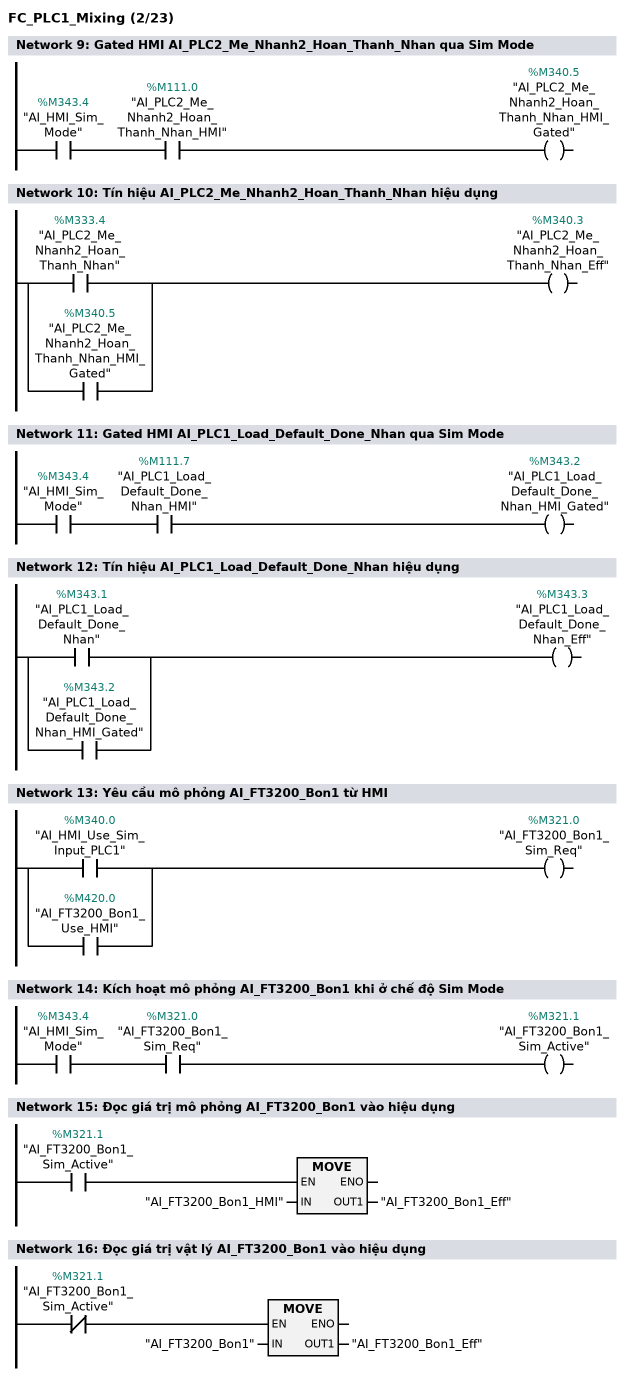
   RUNG wire#powerrail
      Contact( "AI_HMI_Sim_Mode" )
      Contact( "AI_PLC2_Me_Nhanh2_Hoan_Thanh_Nhan_HMI" )
      Coil( "AI_PLC2_Me_Nhanh2_Hoan_Thanh_Nhan_HMI_Gated" )
   END_RUNG
   // the same network as SCL:
   "AI_PLC2_Me_Nhanh2_Hoan_Thanh_Nhan_HMI_Gated" := "AI_HMI_Sim_Mode" AND "AI_PLC2_Me_Nhanh2_Hoan_Thanh_Nhan_HMI";
END_REGION

REGION Network 10: Tín hiệu AI_PLC2_Me_Nhanh2_Hoan_Thanh_Nhan hiệu dụng
   RUNG wire#powerrail
      Contact( "AI_PLC2_Me_Nhanh2_Hoan_Thanh_Nhan" )
      wire#w1
      Coil( "AI_PLC2_Me_Nhanh2_Hoan_Thanh_Nhan_Eff" )
   END_RUNG
   RUNG wire#powerrail
      Contact( "AI_PLC2_Me_Nhanh2_Hoan_Thanh_Nhan_HMI_Gated" )
   END_RUNG wire#w1
   // the same network as SCL:
   "AI_PLC2_Me_Nhanh2_Hoan_Thanh_Nhan_Eff" := "AI_PLC2_Me_Nhanh2_Hoan_Thanh_Nhan" OR "AI_PLC2_Me_Nhanh2_Hoan_Thanh_Nhan_HMI_Gated";
END_REGION

REGION Network 11: Gated HMI AI_PLC1_Load_Default_Done_Nhan qua Sim Mode
   RUNG wire#powerrail
      Contact( "AI_HMI_Sim_Mode" )
      Contact( "AI_PLC1_Load_Default_Done_Nhan_HMI" )
      Coil( "AI_PLC1_Load_Default_Done_Nhan_HMI_Gated" )
   END_RUNG
   // the same network as SCL:
   "AI_PLC1_Load_Default_Done_Nhan_HMI_Gated" := "AI_HMI_Sim_Mode" AND "AI_PLC1_Load_Default_Done_Nhan_HMI";
END_REGION

REGION Network 12: Tín hiệu AI_PLC1_Load_Default_Done_Nhan hiệu dụng
   RUNG wire#powerrail
      Contact( "AI_PLC1_Load_Default_Done_Nhan" )
      wire#w1
      Coil( "AI_PLC1_Load_Default_Done_Nhan_Eff" )
   END_RUNG
   RUNG wire#powerrail
      Contact( "AI_PLC1_Load_Default_Done_Nhan_HMI_Gated" )
   END_RUNG wire#w1
   // the same network as SCL:
   "AI_PLC1_Load_Default_Done_Nhan_Eff" := "AI_PLC1_Load_Default_Done_Nhan" OR "AI_PLC1_Load_Default_Done_Nhan_HMI_Gated";
END_REGION

REGION Network 13: Yêu cầu mô phỏng AI_FT3200_Bon1 từ HMI
   RUNG wire#powerrail
      Contact( "AI_HMI_Use_Sim_Input_PLC1" )
      wire#w1
      Coil( "AI_FT3200_Bon1_Sim_Req" )
   END_RUNG
   RUNG wire#powerrail
      Contact( "AI_FT3200_Bon1_Use_HMI" )
   END_RUNG wire#w1
   // the same network as SCL:
   "AI_FT3200_Bon1_Sim_Req" := "AI_HMI_Use_Sim_Input_PLC1" OR "AI_FT3200_Bon1_Use_HMI";
END_REGION

REGION Network 14: Kích hoạt mô phỏng AI_FT3200_Bon1 khi ở chế độ Sim Mode
   RUNG wire#powerrail
      Contact( "AI_HMI_Sim_Mode" )
      Contact( "AI_FT3200_Bon1_Sim_Req" )
      Coil( "AI_FT3200_Bon1_Sim_Active" )
   END_RUNG
   // the same network as SCL:
   "AI_FT3200_Bon1_Sim_Active" := "AI_HMI_Sim_Mode" AND "AI_FT3200_Bon1_Sim_Req";
END_REGION

REGION Network 15: Đọc giá trị mô phỏng AI_FT3200_Bon1 vào hiệu dụng
   RUNG wire#powerrail
      Contact( "AI_FT3200_Bon1_Sim_Active" )
      { S7_GenerateENO := "TRUE" } Move(in := "AI_FT3200_Bon1_HMI", out1 => "AI_FT3200_Bon1_Eff")
   END_RUNG
   // the same network as SCL:
   IF "AI_FT3200_Bon1_Sim_Active" THEN "AI_FT3200_Bon1_Eff" := "AI_FT3200_Bon1_HMI"; END_IF;
END_REGION

REGION Network 16: Đọc giá trị vật lý AI_FT3200_Bon1 vào hiệu dụng
   RUNG wire#powerrail
      I_Contact( "AI_FT3200_Bon1_Sim_Active" )
      { S7_GenerateENO := "TRUE" } Move(in := "AI_FT3200_Bon1", out1 => "AI_FT3200_Bon1_Eff")
   END_RUNG
   // the same network as SCL:
   IF NOT "AI_FT3200_Bon1_Sim_Active" THEN "AI_FT3200_Bon1_Eff" := "AI_FT3200_Bon1"; END_IF;
END_REGION

REGION Network 17: Yêu cầu mô phỏng AI_FQ3200_Bon1 từ HMI
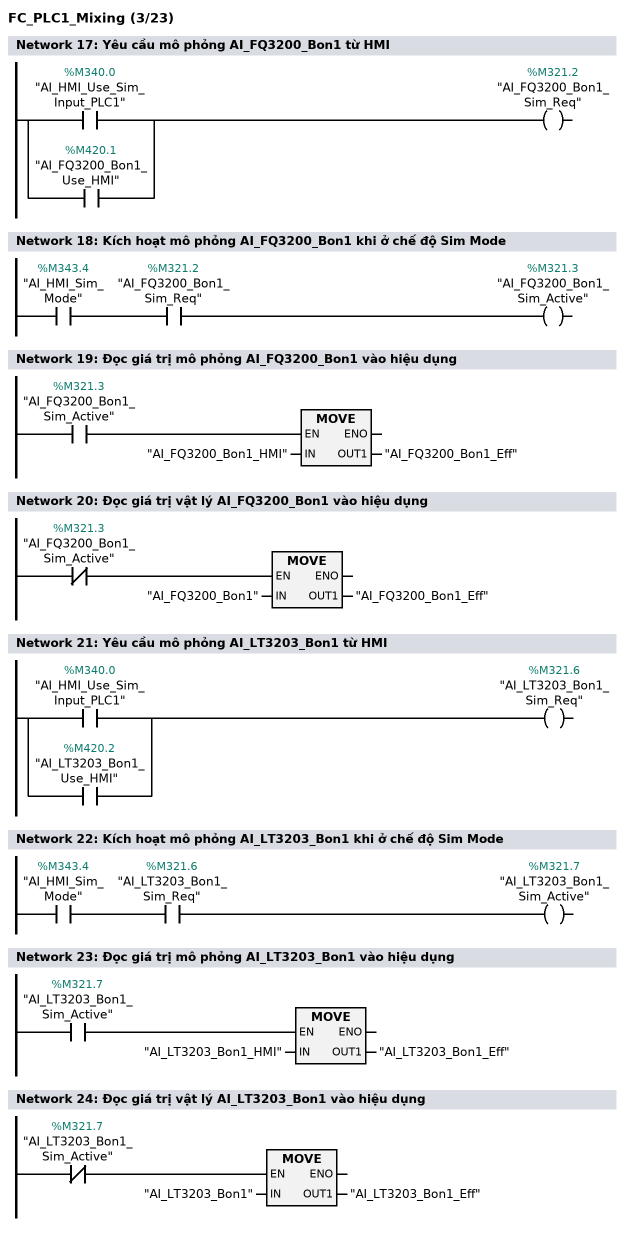
   RUNG wire#powerrail
      Contact( "AI_HMI_Use_Sim_Input_PLC1" )
      wire#w1
      Coil( "AI_FQ3200_Bon1_Sim_Req" )
   END_RUNG
   RUNG wire#powerrail
      Contact( "AI_FQ3200_Bon1_Use_HMI" )
   END_RUNG wire#w1
   // the same network as SCL:
   "AI_FQ3200_Bon1_Sim_Req" := "AI_HMI_Use_Sim_Input_PLC1" OR "AI_FQ3200_Bon1_Use_HMI";
END_REGION

REGION Network 18: Kích hoạt mô phỏng AI_FQ3200_Bon1 khi ở chế độ Sim Mode
   RUNG wire#powerrail
      Contact( "AI_HMI_Sim_Mode" )
      Contact( "AI_FQ3200_Bon1_Sim_Req" )
      Coil( "AI_FQ3200_Bon1_Sim_Active" )
   END_RUNG
   // the same network as SCL:
   "AI_FQ3200_Bon1_Sim_Active" := "AI_HMI_Sim_Mode" AND "AI_FQ3200_Bon1_Sim_Req";
END_REGION

REGION Network 19: Đọc giá trị mô phỏng AI_FQ3200_Bon1 vào hiệu dụng
   RUNG wire#powerrail
      Contact( "AI_FQ3200_Bon1_Sim_Active" )
      { S7_GenerateENO := "TRUE" } Move(in := "AI_FQ3200_Bon1_HMI", out1 => "AI_FQ3200_Bon1_Eff")
   END_RUNG
   // the same network as SCL:
   IF "AI_FQ3200_Bon1_Sim_Active" THEN "AI_FQ3200_Bon1_Eff" := "AI_FQ3200_Bon1_HMI"; END_IF;
END_REGION

REGION Network 20: Đọc giá trị vật lý AI_FQ3200_Bon1 vào hiệu dụng
   RUNG wire#powerrail
      I_Contact( "AI_FQ3200_Bon1_Sim_Active" )
      { S7_GenerateENO := "TRUE" } Move(in := "AI_FQ3200_Bon1", out1 => "AI_FQ3200_Bon1_Eff")
   END_RUNG
   // the same network as SCL:
   IF NOT "AI_FQ3200_Bon1_Sim_Active" THEN "AI_FQ3200_Bon1_Eff" := "AI_FQ3200_Bon1"; END_IF;
END_REGION

REGION Network 21: Yêu cầu mô phỏng AI_LT3203_Bon1 từ HMI
   RUNG wire#powerrail
      Contact( "AI_HMI_Use_Sim_Input_PLC1" )
      wire#w1
      Coil( "AI_LT3203_Bon1_Sim_Req" )
   END_RUNG
   RUNG wire#powerrail
      Contact( "AI_LT3203_Bon1_Use_HMI" )
   END_RUNG wire#w1
   // the same network as SCL:
   "AI_LT3203_Bon1_Sim_Req" := "AI_HMI_Use_Sim_Input_PLC1" OR "AI_LT3203_Bon1_Use_HMI";
END_REGION

REGION Network 22: Kích hoạt mô phỏng AI_LT3203_Bon1 khi ở chế độ Sim Mode
   RUNG wire#powerrail
      Contact( "AI_HMI_Sim_Mode" )
      Contact( "AI_LT3203_Bon1_Sim_Req" )
      Coil( "AI_LT3203_Bon1_Sim_Active" )
   END_RUNG
   // the same network as SCL:
   "AI_LT3203_Bon1_Sim_Active" := "AI_HMI_Sim_Mode" AND "AI_LT3203_Bon1_Sim_Req";
END_REGION

REGION Network 23: Đọc giá trị mô phỏng AI_LT3203_Bon1 vào hiệu dụng
   RUNG wire#powerrail
      Contact( "AI_LT3203_Bon1_Sim_Active" )
      { S7_GenerateENO := "TRUE" } Move(in := "AI_LT3203_Bon1_HMI", out1 => "AI_LT3203_Bon1_Eff")
   END_RUNG
   // the same network as SCL:
   IF "AI_LT3203_Bon1_Sim_Active" THEN "AI_LT3203_Bon1_Eff" := "AI_LT3203_Bon1_HMI"; END_IF;
END_REGION

REGION Network 24: Đọc giá trị vật lý AI_LT3203_Bon1 vào hiệu dụng
   RUNG wire#powerrail
      I_Contact( "AI_LT3203_Bon1_Sim_Active" )
      { S7_GenerateENO := "TRUE" } Move(in := "AI_LT3203_Bon1", out1 => "AI_LT3203_Bon1_Eff")
   END_RUNG
   // the same network as SCL:
   IF NOT "AI_LT3203_Bon1_Sim_Active" THEN "AI_LT3203_Bon1_Eff" := "AI_LT3203_Bon1"; END_IF;
END_REGION

REGION Network 25: Yêu cầu mô phỏng AI_TT3204_Bon1 từ HMI
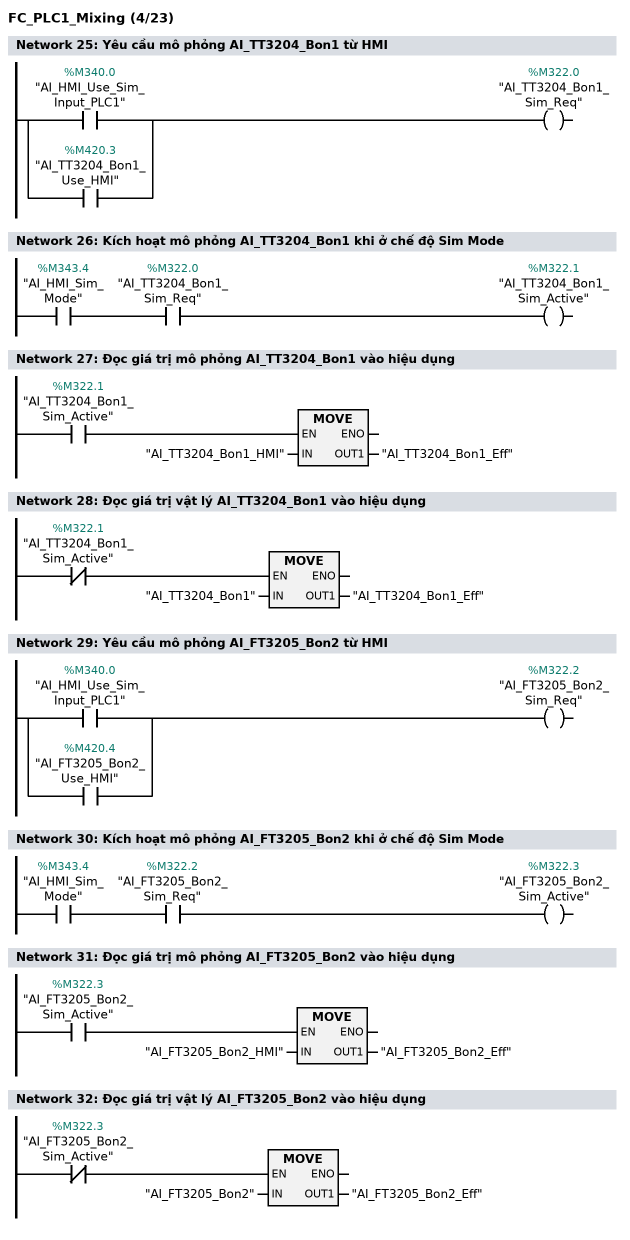
   RUNG wire#powerrail
      Contact( "AI_HMI_Use_Sim_Input_PLC1" )
      wire#w1
      Coil( "AI_TT3204_Bon1_Sim_Req" )
   END_RUNG
   RUNG wire#powerrail
      Contact( "AI_TT3204_Bon1_Use_HMI" )
   END_RUNG wire#w1
   // the same network as SCL:
   "AI_TT3204_Bon1_Sim_Req" := "AI_HMI_Use_Sim_Input_PLC1" OR "AI_TT3204_Bon1_Use_HMI";
END_REGION

REGION Network 26: Kích hoạt mô phỏng AI_TT3204_Bon1 khi ở chế độ Sim Mode
   RUNG wire#powerrail
      Contact( "AI_HMI_Sim_Mode" )
      Contact( "AI_TT3204_Bon1_Sim_Req" )
      Coil( "AI_TT3204_Bon1_Sim_Active" )
   END_RUNG
   // the same network as SCL:
   "AI_TT3204_Bon1_Sim_Active" := "AI_HMI_Sim_Mode" AND "AI_TT3204_Bon1_Sim_Req";
END_REGION

REGION Network 27: Đọc giá trị mô phỏng AI_TT3204_Bon1 vào hiệu dụng
   RUNG wire#powerrail
      Contact( "AI_TT3204_Bon1_Sim_Active" )
      { S7_GenerateENO := "TRUE" } Move(in := "AI_TT3204_Bon1_HMI", out1 => "AI_TT3204_Bon1_Eff")
   END_RUNG
   // the same network as SCL:
   IF "AI_TT3204_Bon1_Sim_Active" THEN "AI_TT3204_Bon1_Eff" := "AI_TT3204_Bon1_HMI"; END_IF;
END_REGION

REGION Network 28: Đọc giá trị vật lý AI_TT3204_Bon1 vào hiệu dụng
   RUNG wire#powerrail
      I_Contact( "AI_TT3204_Bon1_Sim_Active" )
      { S7_GenerateENO := "TRUE" } Move(in := "AI_TT3204_Bon1", out1 => "AI_TT3204_Bon1_Eff")
   END_RUNG
   // the same network as SCL:
   IF NOT "AI_TT3204_Bon1_Sim_Active" THEN "AI_TT3204_Bon1_Eff" := "AI_TT3204_Bon1"; END_IF;
END_REGION

REGION Network 29: Yêu cầu mô phỏng AI_FT3205_Bon2 từ HMI
   RUNG wire#powerrail
      Contact( "AI_HMI_Use_Sim_Input_PLC1" )
      wire#w1
      Coil( "AI_FT3205_Bon2_Sim_Req" )
   END_RUNG
   RUNG wire#powerrail
      Contact( "AI_FT3205_Bon2_Use_HMI" )
   END_RUNG wire#w1
   // the same network as SCL:
   "AI_FT3205_Bon2_Sim_Req" := "AI_HMI_Use_Sim_Input_PLC1" OR "AI_FT3205_Bon2_Use_HMI";
END_REGION

REGION Network 30: Kích hoạt mô phỏng AI_FT3205_Bon2 khi ở chế độ Sim Mode
   RUNG wire#powerrail
      Contact( "AI_HMI_Sim_Mode" )
      Contact( "AI_FT3205_Bon2_Sim_Req" )
      Coil( "AI_FT3205_Bon2_Sim_Active" )
   END_RUNG
   // the same network as SCL:
   "AI_FT3205_Bon2_Sim_Active" := "AI_HMI_Sim_Mode" AND "AI_FT3205_Bon2_Sim_Req";
END_REGION

REGION Network 31: Đọc giá trị mô phỏng AI_FT3205_Bon2 vào hiệu dụng
   RUNG wire#powerrail
      Contact( "AI_FT3205_Bon2_Sim_Active" )
      { S7_GenerateENO := "TRUE" } Move(in := "AI_FT3205_Bon2_HMI", out1 => "AI_FT3205_Bon2_Eff")
   END_RUNG
   // the same network as SCL:
   IF "AI_FT3205_Bon2_Sim_Active" THEN "AI_FT3205_Bon2_Eff" := "AI_FT3205_Bon2_HMI"; END_IF;
END_REGION

REGION Network 32: Đọc giá trị vật lý AI_FT3205_Bon2 vào hiệu dụng
   RUNG wire#powerrail
      I_Contact( "AI_FT3205_Bon2_Sim_Active" )
      { S7_GenerateENO := "TRUE" } Move(in := "AI_FT3205_Bon2", out1 => "AI_FT3205_Bon2_Eff")
   END_RUNG
   // the same network as SCL:
   IF NOT "AI_FT3205_Bon2_Sim_Active" THEN "AI_FT3205_Bon2_Eff" := "AI_FT3205_Bon2"; END_IF;
END_REGION

REGION Network 33: Yêu cầu mô phỏng AI_FQ3205_Bon2 từ HMI
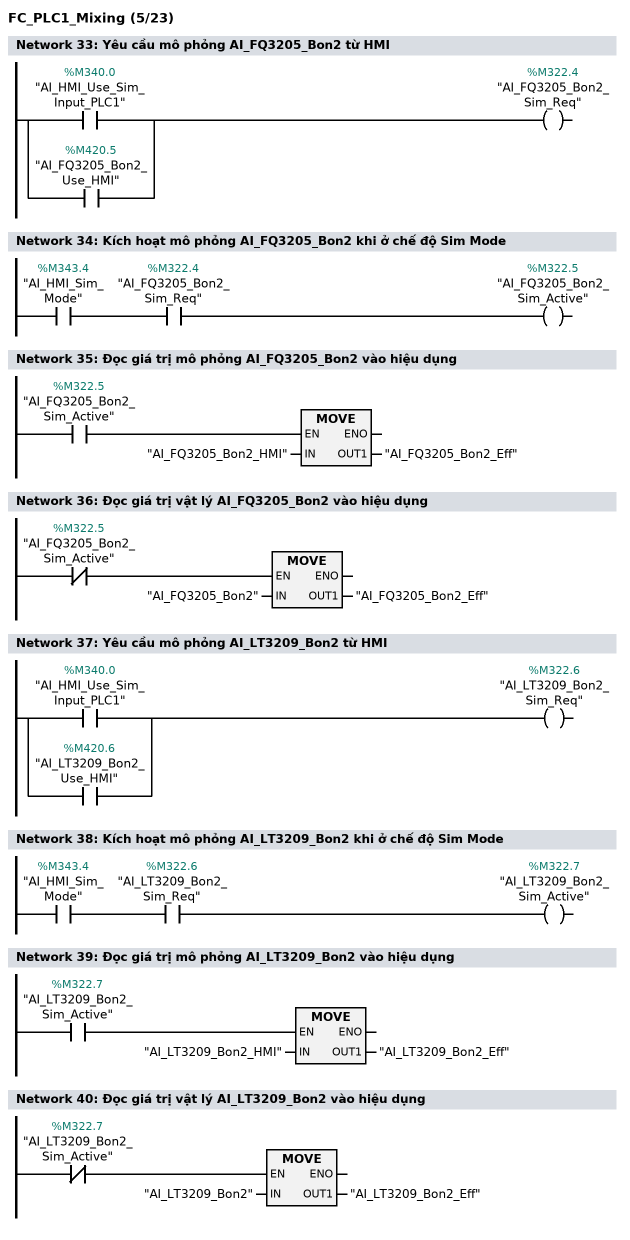
   RUNG wire#powerrail
      Contact( "AI_HMI_Use_Sim_Input_PLC1" )
      wire#w1
      Coil( "AI_FQ3205_Bon2_Sim_Req" )
   END_RUNG
   RUNG wire#powerrail
      Contact( "AI_FQ3205_Bon2_Use_HMI" )
   END_RUNG wire#w1
   // the same network as SCL:
   "AI_FQ3205_Bon2_Sim_Req" := "AI_HMI_Use_Sim_Input_PLC1" OR "AI_FQ3205_Bon2_Use_HMI";
END_REGION

REGION Network 34: Kích hoạt mô phỏng AI_FQ3205_Bon2 khi ở chế độ Sim Mode
   RUNG wire#powerrail
      Contact( "AI_HMI_Sim_Mode" )
      Contact( "AI_FQ3205_Bon2_Sim_Req" )
      Coil( "AI_FQ3205_Bon2_Sim_Active" )
   END_RUNG
   // the same network as SCL:
   "AI_FQ3205_Bon2_Sim_Active" := "AI_HMI_Sim_Mode" AND "AI_FQ3205_Bon2_Sim_Req";
END_REGION

REGION Network 35: Đọc giá trị mô phỏng AI_FQ3205_Bon2 vào hiệu dụng
   RUNG wire#powerrail
      Contact( "AI_FQ3205_Bon2_Sim_Active" )
      { S7_GenerateENO := "TRUE" } Move(in := "AI_FQ3205_Bon2_HMI", out1 => "AI_FQ3205_Bon2_Eff")
   END_RUNG
   // the same network as SCL:
   IF "AI_FQ3205_Bon2_Sim_Active" THEN "AI_FQ3205_Bon2_Eff" := "AI_FQ3205_Bon2_HMI"; END_IF;
END_REGION

REGION Network 36: Đọc giá trị vật lý AI_FQ3205_Bon2 vào hiệu dụng
   RUNG wire#powerrail
      I_Contact( "AI_FQ3205_Bon2_Sim_Active" )
      { S7_GenerateENO := "TRUE" } Move(in := "AI_FQ3205_Bon2", out1 => "AI_FQ3205_Bon2_Eff")
   END_RUNG
   // the same network as SCL:
   IF NOT "AI_FQ3205_Bon2_Sim_Active" THEN "AI_FQ3205_Bon2_Eff" := "AI_FQ3205_Bon2"; END_IF;
END_REGION

REGION Network 37: Yêu cầu mô phỏng AI_LT3209_Bon2 từ HMI
   RUNG wire#powerrail
      Contact( "AI_HMI_Use_Sim_Input_PLC1" )
      wire#w1
      Coil( "AI_LT3209_Bon2_Sim_Req" )
   END_RUNG
   RUNG wire#powerrail
      Contact( "AI_LT3209_Bon2_Use_HMI" )
   END_RUNG wire#w1
   // the same network as SCL:
   "AI_LT3209_Bon2_Sim_Req" := "AI_HMI_Use_Sim_Input_PLC1" OR "AI_LT3209_Bon2_Use_HMI";
END_REGION

REGION Network 38: Kích hoạt mô phỏng AI_LT3209_Bon2 khi ở chế độ Sim Mode
   RUNG wire#powerrail
      Contact( "AI_HMI_Sim_Mode" )
      Contact( "AI_LT3209_Bon2_Sim_Req" )
      Coil( "AI_LT3209_Bon2_Sim_Active" )
   END_RUNG
   // the same network as SCL:
   "AI_LT3209_Bon2_Sim_Active" := "AI_HMI_Sim_Mode" AND "AI_LT3209_Bon2_Sim_Req";
END_REGION

REGION Network 39: Đọc giá trị mô phỏng AI_LT3209_Bon2 vào hiệu dụng
   RUNG wire#powerrail
      Contact( "AI_LT3209_Bon2_Sim_Active" )
      { S7_GenerateENO := "TRUE" } Move(in := "AI_LT3209_Bon2_HMI", out1 => "AI_LT3209_Bon2_Eff")
   END_RUNG
   // the same network as SCL:
   IF "AI_LT3209_Bon2_Sim_Active" THEN "AI_LT3209_Bon2_Eff" := "AI_LT3209_Bon2_HMI"; END_IF;
END_REGION

REGION Network 40: Đọc giá trị vật lý AI_LT3209_Bon2 vào hiệu dụng
   RUNG wire#powerrail
      I_Contact( "AI_LT3209_Bon2_Sim_Active" )
      { S7_GenerateENO := "TRUE" } Move(in := "AI_LT3209_Bon2", out1 => "AI_LT3209_Bon2_Eff")
   END_RUNG
   // the same network as SCL:
   IF NOT "AI_LT3209_Bon2_Sim_Active" THEN "AI_LT3209_Bon2_Eff" := "AI_LT3209_Bon2"; END_IF;
END_REGION

REGION Network 41: Yêu cầu mô phỏng AI_TT3208_Bon2 từ HMI
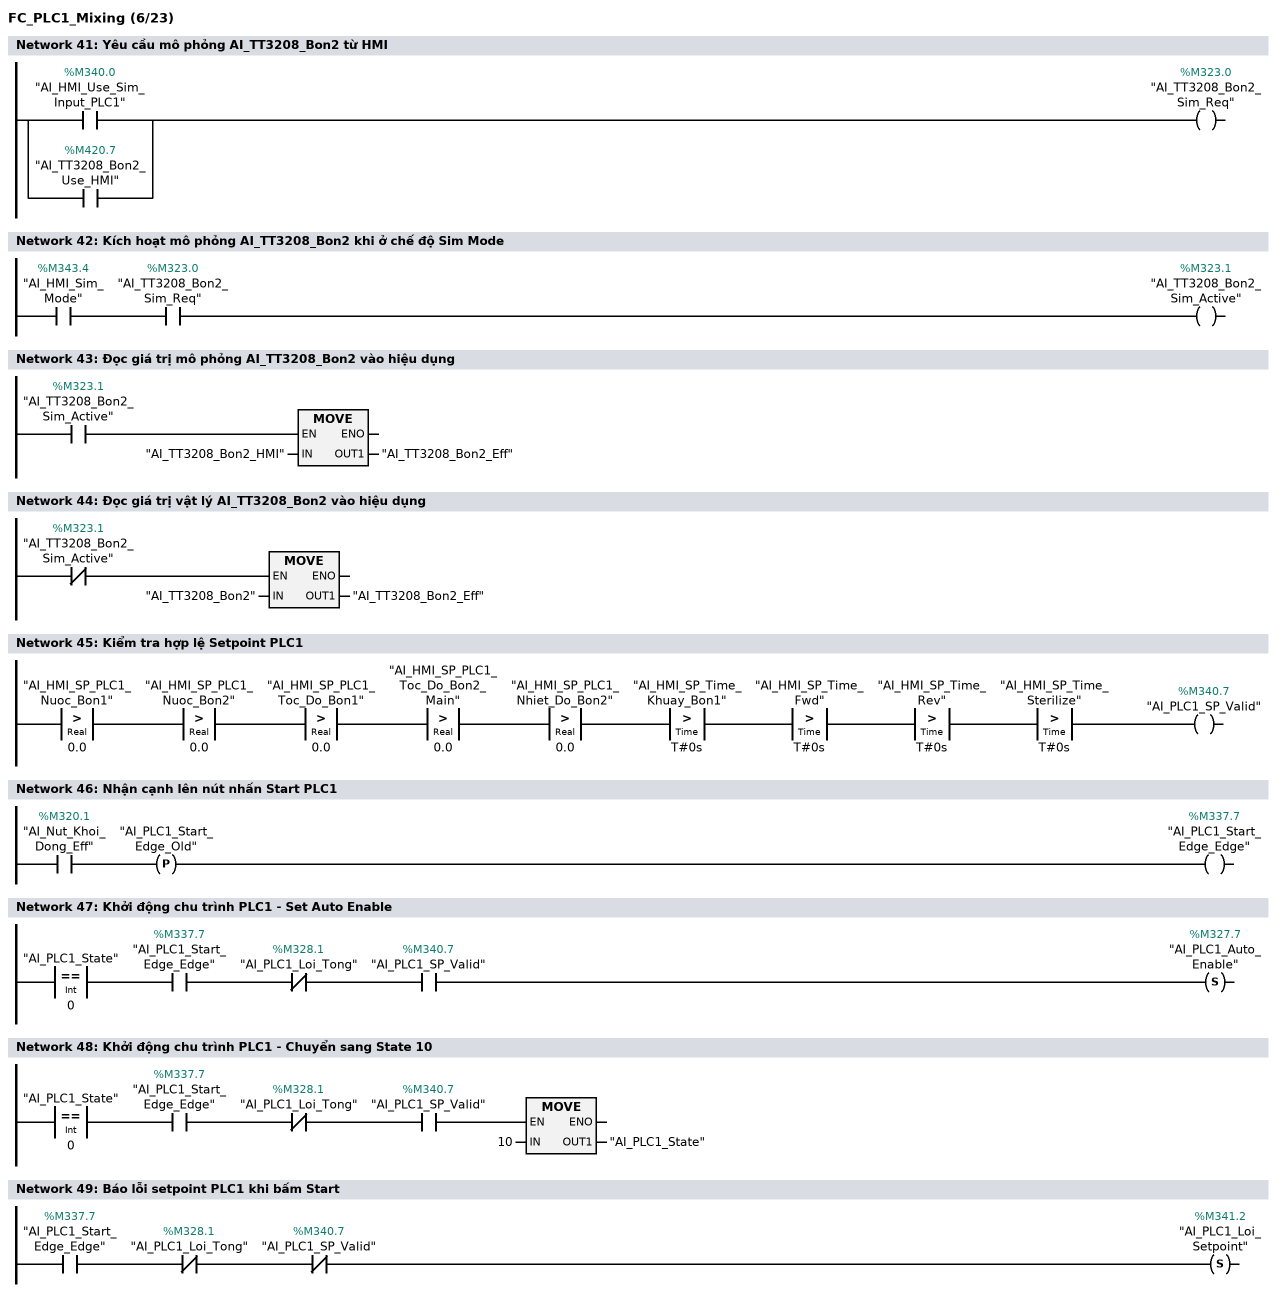
   RUNG wire#powerrail
      Contact( "AI_HMI_Use_Sim_Input_PLC1" )
      wire#w1
      Coil( "AI_TT3208_Bon2_Sim_Req" )
   END_RUNG
   RUNG wire#powerrail
      Contact( "AI_TT3208_Bon2_Use_HMI" )
   END_RUNG wire#w1
   // the same network as SCL:
   "AI_TT3208_Bon2_Sim_Req" := "AI_HMI_Use_Sim_Input_PLC1" OR "AI_TT3208_Bon2_Use_HMI";
END_REGION

REGION Network 42: Kích hoạt mô phỏng AI_TT3208_Bon2 khi ở chế độ Sim Mode
   RUNG wire#powerrail
      Contact( "AI_HMI_Sim_Mode" )
      Contact( "AI_TT3208_Bon2_Sim_Req" )
      Coil( "AI_TT3208_Bon2_Sim_Active" )
   END_RUNG
   // the same network as SCL:
   "AI_TT3208_Bon2_Sim_Active" := "AI_HMI_Sim_Mode" AND "AI_TT3208_Bon2_Sim_Req";
END_REGION

REGION Network 43: Đọc giá trị mô phỏng AI_TT3208_Bon2 vào hiệu dụng
   RUNG wire#powerrail
      Contact( "AI_TT3208_Bon2_Sim_Active" )
      { S7_GenerateENO := "TRUE" } Move(in := "AI_TT3208_Bon2_HMI", out1 => "AI_TT3208_Bon2_Eff")
   END_RUNG
   // the same network as SCL:
   IF "AI_TT3208_Bon2_Sim_Active" THEN "AI_TT3208_Bon2_Eff" := "AI_TT3208_Bon2_HMI"; END_IF;
END_REGION

REGION Network 44: Đọc giá trị vật lý AI_TT3208_Bon2 vào hiệu dụng
   RUNG wire#powerrail
      I_Contact( "AI_TT3208_Bon2_Sim_Active" )
      { S7_GenerateENO := "TRUE" } Move(in := "AI_TT3208_Bon2", out1 => "AI_TT3208_Bon2_Eff")
   END_RUNG
   // the same network as SCL:
   IF NOT "AI_TT3208_Bon2_Sim_Active" THEN "AI_TT3208_Bon2_Eff" := "AI_TT3208_Bon2"; END_IF;
END_REGION

REGION Network 45: Kiểm tra hợp lệ Setpoint PLC1
   RUNG wire#powerrail
      { S7_Templates := "SrcType := Real" } GT_Contact(in1 := "AI_HMI_SP_PLC1_Nuoc_Bon1", in2 := 0.0)
      { S7_Templates := "SrcType := Real" } GT_Contact(in1 := "AI_HMI_SP_PLC1_Nuoc_Bon2", in2 := 0.0)
      { S7_Templates := "SrcType := Real" } GT_Contact(in1 := "AI_HMI_SP_PLC1_Toc_Do_Bon1", in2 := 0.0)
      { S7_Templates := "SrcType := Real" } GT_Contact(in1 := "AI_HMI_SP_PLC1_Toc_Do_Bon2_Main", in2 := 0.0)
      { S7_Templates := "SrcType := Real" } GT_Contact(in1 := "AI_HMI_SP_PLC1_Nhiet_Do_Bon2", in2 := 0.0)
      { S7_Templates := "SrcType := Time" } GT_Contact(in1 := "AI_HMI_SP_Time_Khuay_Bon1", in2 := T#0s)
      { S7_Templates := "SrcType := Time" } GT_Contact(in1 := "AI_HMI_SP_Time_Fwd", in2 := T#0s)
      { S7_Templates := "SrcType := Time" } GT_Contact(in1 := "AI_HMI_SP_Time_Rev", in2 := T#0s)
      { S7_Templates := "SrcType := Time" } GT_Contact(in1 := "AI_HMI_SP_Time_Sterilize", in2 := T#0s)
      Coil( "AI_PLC1_SP_Valid" )
   END_RUNG
   // the same network as SCL:
   "AI_PLC1_SP_Valid" := ("AI_HMI_SP_PLC1_Nuoc_Bon1" > 0.0) AND ("AI_HMI_SP_PLC1_Nuoc_Bon2" > 0.0) AND ("AI_HMI_SP_PLC1_Toc_Do_Bon1" > 0.0) AND ("AI_HMI_SP_PLC1_Toc_Do_Bon2_Main" > 0.0) AND ("AI_HMI_SP_PLC1_Nhiet_Do_Bon2" > 0.0) AND ("AI_HMI_SP_Time_Khuay_Bon1" > T#0s) AND ("AI_HMI_SP_Time_Fwd" > T#0s) AND ("AI_HMI_SP_Time_Rev" > T#0s) AND ("AI_HMI_SP_Time_Sterilize" > T#0s);
END_REGION

REGION Network 46: Nhận cạnh lên nút nhấn Start PLC1
   RUNG wire#powerrail
      Contact( "AI_Nut_Khoi_Dong_Eff" )
      P_Trig( "AI_PLC1_Start_Edge_Old" )
      Coil( "AI_PLC1_Start_Edge_Edge" )
   END_RUNG
   // the same network as SCL:
   #_w1 := "AI_Nut_Khoi_Dong_Eff" AND NOT "AI_PLC1_Start_Edge_Old";   // rising edge
   "AI_PLC1_Start_Edge_Old" := "AI_Nut_Khoi_Dong_Eff";
   "AI_PLC1_Start_Edge_Edge" := #_w1;
END_REGION

REGION Network 47: Khởi động chu trình PLC1 - Set Auto Enable
   RUNG wire#powerrail
      { S7_Templates := "SrcType := Int" } EQ_Contact(in1 := "AI_PLC1_State", in2 := 0)
      Contact( "AI_PLC1_Start_Edge_Edge" )
      I_Contact( "AI_PLC1_Loi_Tong" )
      Contact( "AI_PLC1_SP_Valid" )
      S_Coil( "AI_PLC1_Auto_Enable" )
   END_RUNG
   // the same network as SCL:
   IF ("AI_PLC1_State" = 0) AND "AI_PLC1_Start_Edge_Edge" AND NOT "AI_PLC1_Loi_Tong" AND "AI_PLC1_SP_Valid" THEN
       "AI_PLC1_Auto_Enable" := TRUE;
   END_IF;
END_REGION

REGION Network 48: Khởi động chu trình PLC1 - Chuyển sang State 10
   RUNG wire#powerrail
      { S7_Templates := "SrcType := Int" } EQ_Contact(in1 := "AI_PLC1_State", in2 := 0)
      Contact( "AI_PLC1_Start_Edge_Edge" )
      I_Contact( "AI_PLC1_Loi_Tong" )
      Contact( "AI_PLC1_SP_Valid" )
      { S7_GenerateENO := "TRUE" } Move(in := 10, out1 => "AI_PLC1_State")
   END_RUNG
   // the same network as SCL:
   IF ("AI_PLC1_State" = 0) AND "AI_PLC1_Start_Edge_Edge" AND NOT "AI_PLC1_Loi_Tong" AND "AI_PLC1_SP_Valid" THEN
       "AI_PLC1_State" := 10;
   END_IF;
END_REGION

REGION Network 49: Báo lỗi setpoint PLC1 khi bấm Start
   RUNG wire#powerrail
      Contact( "AI_PLC1_Start_Edge_Edge" )
      I_Contact( "AI_PLC1_Loi_Tong" )
      I_Contact( "AI_PLC1_SP_Valid" )
      S_Coil( "AI_PLC1_Loi_Setpoint" )
   END_RUNG
   // the same network as SCL:
   IF "AI_PLC1_Start_Edge_Edge" AND NOT "AI_PLC1_Loi_Tong" AND NOT "AI_PLC1_SP_Valid" THEN
       "AI_PLC1_Loi_Setpoint" := TRUE;
   END_IF;
END_REGION

REGION Network 50: Stop PLC1 từ nút vật lý hoặc HMI
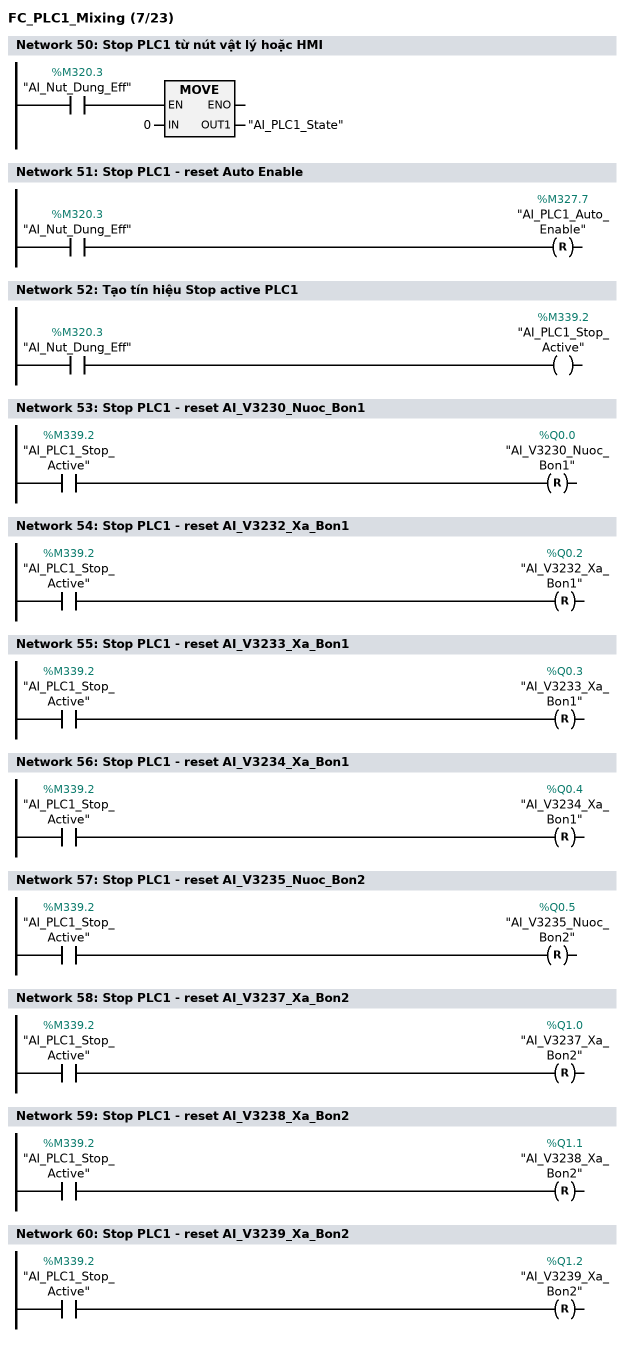
   RUNG wire#powerrail
      Contact( "AI_Nut_Dung_Eff" )
      { S7_GenerateENO := "TRUE" } Move(in := 0, out1 => "AI_PLC1_State")
   END_RUNG
   // the same network as SCL:
   IF "AI_Nut_Dung_Eff" THEN "AI_PLC1_State" := 0; END_IF;
END_REGION

REGION Network 51: Stop PLC1 - reset Auto Enable
   RUNG wire#powerrail
      Contact( "AI_Nut_Dung_Eff" )
      R_Coil( "AI_PLC1_Auto_Enable" )
   END_RUNG
   // the same network as SCL:
   IF "AI_Nut_Dung_Eff" THEN "AI_PLC1_Auto_Enable" := FALSE; END_IF;
END_REGION

REGION Network 52: Tạo tín hiệu Stop active PLC1
   RUNG wire#powerrail
      Contact( "AI_Nut_Dung_Eff" )
      Coil( "AI_PLC1_Stop_Active" )
   END_RUNG
   // the same network as SCL:
   "AI_PLC1_Stop_Active" := "AI_Nut_Dung_Eff";
END_REGION

REGION Network 53: Stop PLC1 - reset AI_V3230_Nuoc_Bon1
   RUNG wire#powerrail
      Contact( "AI_PLC1_Stop_Active" )
      R_Coil( "AI_V3230_Nuoc_Bon1" )
   END_RUNG
   // the same network as SCL:
   IF "AI_PLC1_Stop_Active" THEN "AI_V3230_Nuoc_Bon1" := FALSE; END_IF;
END_REGION

REGION Network 54: Stop PLC1 - reset AI_V3232_Xa_Bon1
   RUNG wire#powerrail
      Contact( "AI_PLC1_Stop_Active" )
      R_Coil( "AI_V3232_Xa_Bon1" )
   END_RUNG
   // the same network as SCL:
   IF "AI_PLC1_Stop_Active" THEN "AI_V3232_Xa_Bon1" := FALSE; END_IF;
END_REGION

REGION Network 55: Stop PLC1 - reset AI_V3233_Xa_Bon1
   RUNG wire#powerrail
      Contact( "AI_PLC1_Stop_Active" )
      R_Coil( "AI_V3233_Xa_Bon1" )
   END_RUNG
   // the same network as SCL:
   IF "AI_PLC1_Stop_Active" THEN "AI_V3233_Xa_Bon1" := FALSE; END_IF;
END_REGION

REGION Network 56: Stop PLC1 - reset AI_V3234_Xa_Bon1
   RUNG wire#powerrail
      Contact( "AI_PLC1_Stop_Active" )
      R_Coil( "AI_V3234_Xa_Bon1" )
   END_RUNG
   // the same network as SCL:
   IF "AI_PLC1_Stop_Active" THEN "AI_V3234_Xa_Bon1" := FALSE; END_IF;
END_REGION

REGION Network 57: Stop PLC1 - reset AI_V3235_Nuoc_Bon2
   RUNG wire#powerrail
      Contact( "AI_PLC1_Stop_Active" )
      R_Coil( "AI_V3235_Nuoc_Bon2" )
   END_RUNG
   // the same network as SCL:
   IF "AI_PLC1_Stop_Active" THEN "AI_V3235_Nuoc_Bon2" := FALSE; END_IF;
END_REGION

REGION Network 58: Stop PLC1 - reset AI_V3237_Xa_Bon2
   RUNG wire#powerrail
      Contact( "AI_PLC1_Stop_Active" )
      R_Coil( "AI_V3237_Xa_Bon2" )
   END_RUNG
   // the same network as SCL:
   IF "AI_PLC1_Stop_Active" THEN "AI_V3237_Xa_Bon2" := FALSE; END_IF;
END_REGION

REGION Network 59: Stop PLC1 - reset AI_V3238_Xa_Bon2
   RUNG wire#powerrail
      Contact( "AI_PLC1_Stop_Active" )
      R_Coil( "AI_V3238_Xa_Bon2" )
   END_RUNG
   // the same network as SCL:
   IF "AI_PLC1_Stop_Active" THEN "AI_V3238_Xa_Bon2" := FALSE; END_IF;
END_REGION

REGION Network 60: Stop PLC1 - reset AI_V3239_Xa_Bon2
   RUNG wire#powerrail
      Contact( "AI_PLC1_Stop_Active" )
      R_Coil( "AI_V3239_Xa_Bon2" )
   END_RUNG
   // the same network as SCL:
   IF "AI_PLC1_Stop_Active" THEN "AI_V3239_Xa_Bon2" := FALSE; END_IF;
END_REGION

REGION Network 61: Stop PLC1 - reset AI_Pump3264_Chuyen_Nhanh1
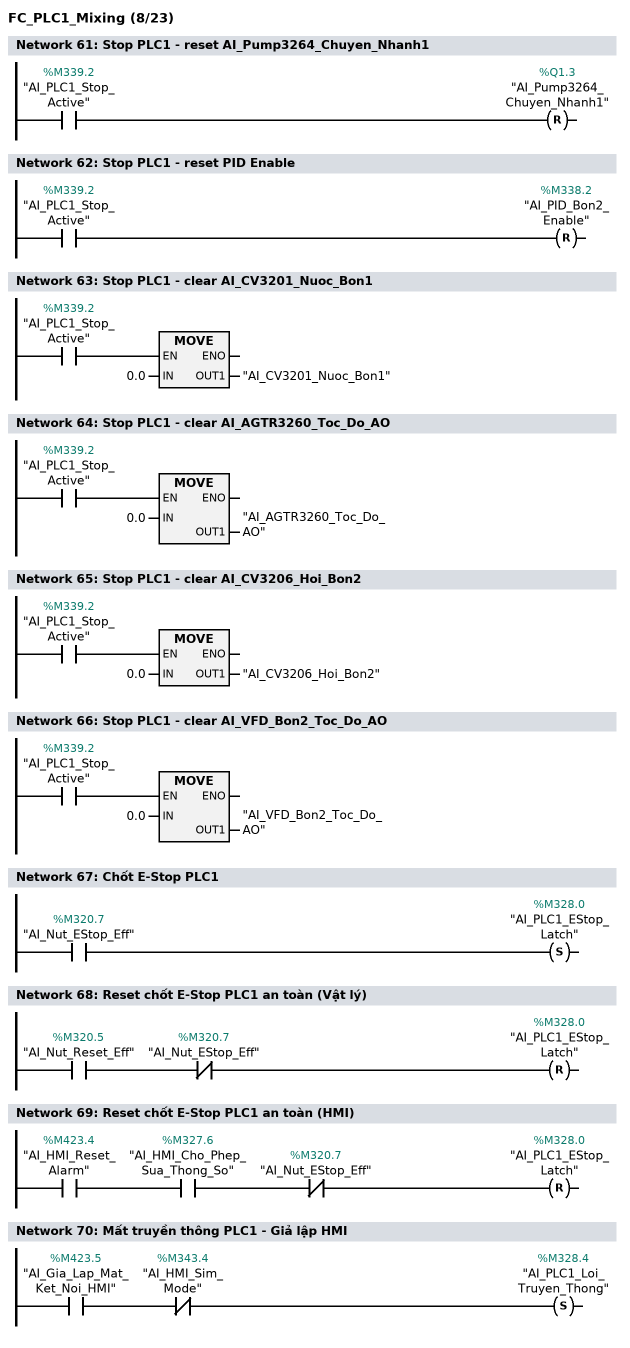
   RUNG wire#powerrail
      Contact( "AI_PLC1_Stop_Active" )
      R_Coil( "AI_Pump3264_Chuyen_Nhanh1" )
   END_RUNG
   // the same network as SCL:
   IF "AI_PLC1_Stop_Active" THEN "AI_Pump3264_Chuyen_Nhanh1" := FALSE; END_IF;
END_REGION

REGION Network 62: Stop PLC1 - reset PID Enable
   RUNG wire#powerrail
      Contact( "AI_PLC1_Stop_Active" )
      R_Coil( "AI_PID_Bon2_Enable" )
   END_RUNG
   // the same network as SCL:
   IF "AI_PLC1_Stop_Active" THEN "AI_PID_Bon2_Enable" := FALSE; END_IF;
END_REGION

REGION Network 63: Stop PLC1 - clear AI_CV3201_Nuoc_Bon1
   RUNG wire#powerrail
      Contact( "AI_PLC1_Stop_Active" )
      { S7_GenerateENO := "TRUE" } Move(in := 0.0, out1 => "AI_CV3201_Nuoc_Bon1")
   END_RUNG
   // the same network as SCL:
   IF "AI_PLC1_Stop_Active" THEN "AI_CV3201_Nuoc_Bon1" := 0.0; END_IF;
END_REGION

REGION Network 64: Stop PLC1 - clear AI_AGTR3260_Toc_Do_AO
   RUNG wire#powerrail
      Contact( "AI_PLC1_Stop_Active" )
      { S7_GenerateENO := "TRUE" } Move(in := 0.0, out1 => "AI_AGTR3260_Toc_Do_AO")
   END_RUNG
   // the same network as SCL:
   IF "AI_PLC1_Stop_Active" THEN "AI_AGTR3260_Toc_Do_AO" := 0.0; END_IF;
END_REGION

REGION Network 65: Stop PLC1 - clear AI_CV3206_Hoi_Bon2
   RUNG wire#powerrail
      Contact( "AI_PLC1_Stop_Active" )
      { S7_GenerateENO := "TRUE" } Move(in := 0.0, out1 => "AI_CV3206_Hoi_Bon2")
   END_RUNG
   // the same network as SCL:
   IF "AI_PLC1_Stop_Active" THEN "AI_CV3206_Hoi_Bon2" := 0.0; END_IF;
END_REGION

REGION Network 66: Stop PLC1 - clear AI_VFD_Bon2_Toc_Do_AO
   RUNG wire#powerrail
      Contact( "AI_PLC1_Stop_Active" )
      { S7_GenerateENO := "TRUE" } Move(in := 0.0, out1 => "AI_VFD_Bon2_Toc_Do_AO")
   END_RUNG
   // the same network as SCL:
   IF "AI_PLC1_Stop_Active" THEN "AI_VFD_Bon2_Toc_Do_AO" := 0.0; END_IF;
END_REGION

REGION Network 67: Chốt E-Stop PLC1
   RUNG wire#powerrail
      Contact( "AI_Nut_EStop_Eff" )
      S_Coil( "AI_PLC1_EStop_Latch" )
   END_RUNG
   // the same network as SCL:
   IF "AI_Nut_EStop_Eff" THEN "AI_PLC1_EStop_Latch" := TRUE; END_IF;
END_REGION

REGION Network 68: Reset chốt E-Stop PLC1 an toàn (Vật lý)
   RUNG wire#powerrail
      Contact( "AI_Nut_Reset_Eff" )
      I_Contact( "AI_Nut_EStop_Eff" )
      R_Coil( "AI_PLC1_EStop_Latch" )
   END_RUNG
   // the same network as SCL:
   IF "AI_Nut_Reset_Eff" AND NOT "AI_Nut_EStop_Eff" THEN "AI_PLC1_EStop_Latch" := FALSE; END_IF;
END_REGION

REGION Network 69: Reset chốt E-Stop PLC1 an toàn (HMI)
   RUNG wire#powerrail
      Contact( "AI_HMI_Reset_Alarm" )
      Contact( "AI_HMI_Cho_Phep_Sua_Thong_So" )
      I_Contact( "AI_Nut_EStop_Eff" )
      R_Coil( "AI_PLC1_EStop_Latch" )
   END_RUNG
   // the same network as SCL:
   IF "AI_HMI_Reset_Alarm" AND "AI_HMI_Cho_Phep_Sua_Thong_So" AND NOT "AI_Nut_EStop_Eff" THEN
       "AI_PLC1_EStop_Latch" := FALSE;
   END_IF;
END_REGION

REGION Network 70: Mất truyền thông PLC1 - Giả lập HMI
   RUNG wire#powerrail
      Contact( "AI_Gia_Lap_Mat_Ket_Noi_HMI" )
      I_Contact( "AI_HMI_Sim_Mode" )
      S_Coil( "AI_PLC1_Loi_Truyen_Thong" )
   END_RUNG
   // the same network as SCL:
   IF "AI_Gia_Lap_Mat_Ket_Noi_HMI" AND NOT "AI_HMI_Sim_Mode" THEN "AI_PLC1_Loi_Truyen_Thong" := TRUE; END_IF;
END_REGION

REGION Network 71: Mất truyền thông PLC1 - Heartbeat Timeout
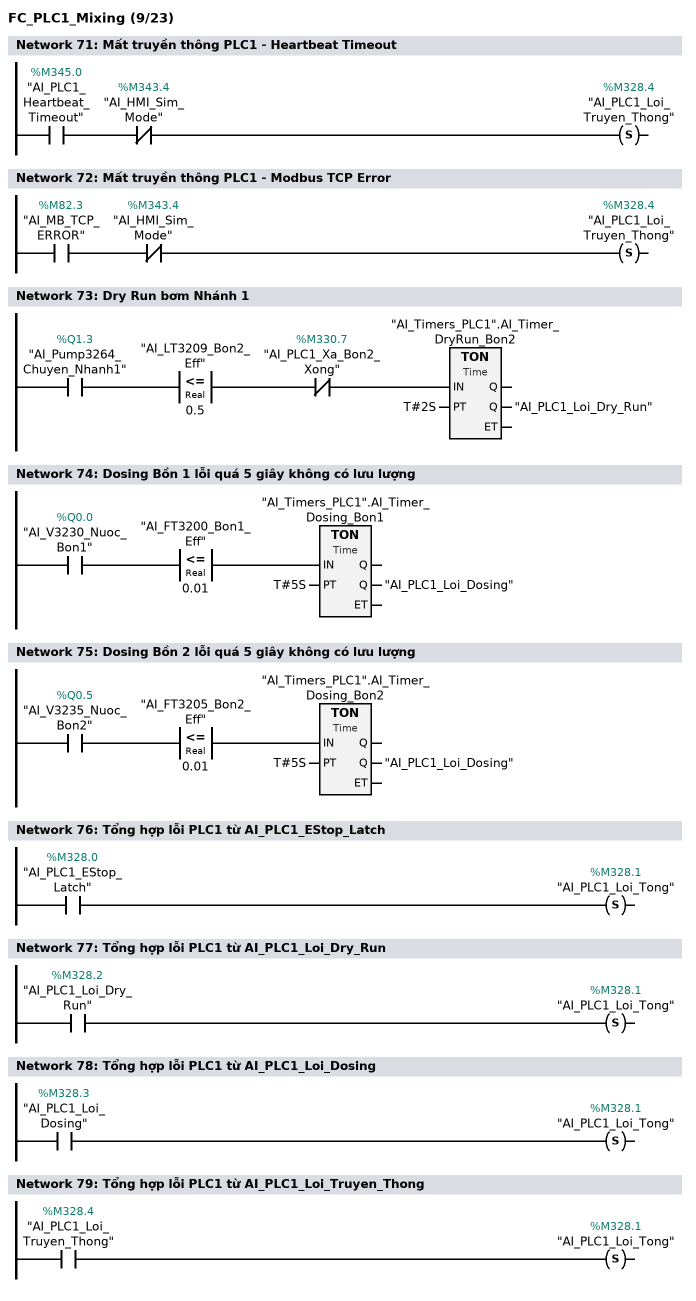
   RUNG wire#powerrail
      Contact( "AI_PLC1_Heartbeat_Timeout" )
      I_Contact( "AI_HMI_Sim_Mode" )
      S_Coil( "AI_PLC1_Loi_Truyen_Thong" )
   END_RUNG
   // the same network as SCL:
   IF "AI_PLC1_Heartbeat_Timeout" AND NOT "AI_HMI_Sim_Mode" THEN "AI_PLC1_Loi_Truyen_Thong" := TRUE; END_IF;
END_REGION

REGION Network 72: Mất truyền thông PLC1 - Modbus TCP Error
   RUNG wire#powerrail
      Contact( "AI_MB_TCP_ERROR" )
      I_Contact( "AI_HMI_Sim_Mode" )
      S_Coil( "AI_PLC1_Loi_Truyen_Thong" )
   END_RUNG
   // the same network as SCL:
   IF "AI_MB_TCP_ERROR" AND NOT "AI_HMI_Sim_Mode" THEN "AI_PLC1_Loi_Truyen_Thong" := TRUE; END_IF;
END_REGION

REGION Network 73: Dry Run bơm Nhánh 1
   RUNG wire#powerrail
      Contact( "AI_Pump3264_Chuyen_Nhanh1" )
      { S7_Templates := "SrcType := Real" } LE_Contact(in1 := "AI_LT3209_Bon2_Eff", in2 := 0.5)
      I_Contact( "AI_PLC1_Xa_Bon2_Xong" )
      { S7_Templates := "time_type := Time" } "AI_Timers_PLC1".AI_Timer_DryRun_Bon2.TON(pt := T#2S, q => "AI_PLC1_Loi_Dry_Run", et =>)
   END_RUNG
   // the same network as SCL:
   "AI_Timers_PLC1".AI_Timer_DryRun_Bon2.TON(IN := "AI_Pump3264_Chuyen_Nhanh1" AND ("AI_LT3209_Bon2_Eff" <= 0.5) AND NOT "AI_PLC1_Xa_Bon2_Xong",
                           PT := T#2S,
                           Q => "AI_PLC1_Loi_Dry_Run");
END_REGION

REGION Network 74: Dosing Bồn 1 lỗi quá 5 giây không có lưu lượng
   RUNG wire#powerrail
      Contact( "AI_V3230_Nuoc_Bon1" )
      { S7_Templates := "SrcType := Real" } LE_Contact(in1 := "AI_FT3200_Bon1_Eff", in2 := 0.01)
      { S7_Templates := "time_type := Time" } "AI_Timers_PLC1".AI_Timer_Dosing_Bon1.TON(pt := T#5S, q => "AI_PLC1_Loi_Dosing", et =>)
   END_RUNG
   // the same network as SCL:
   "AI_Timers_PLC1".AI_Timer_Dosing_Bon1.TON(IN := "AI_V3230_Nuoc_Bon1" AND ("AI_FT3200_Bon1_Eff" <= 0.01),
                           PT := T#5S,
                           Q => "AI_PLC1_Loi_Dosing");
END_REGION

REGION Network 75: Dosing Bồn 2 lỗi quá 5 giây không có lưu lượng
   RUNG wire#powerrail
      Contact( "AI_V3235_Nuoc_Bon2" )
      { S7_Templates := "SrcType := Real" } LE_Contact(in1 := "AI_FT3205_Bon2_Eff", in2 := 0.01)
      { S7_Templates := "time_type := Time" } "AI_Timers_PLC1".AI_Timer_Dosing_Bon2.TON(pt := T#5S, q => "AI_PLC1_Loi_Dosing", et =>)
   END_RUNG
   // the same network as SCL:
   "AI_Timers_PLC1".AI_Timer_Dosing_Bon2.TON(IN := "AI_V3235_Nuoc_Bon2" AND ("AI_FT3205_Bon2_Eff" <= 0.01),
                           PT := T#5S,
                           Q => "AI_PLC1_Loi_Dosing");
END_REGION

REGION Network 76: Tổng hợp lỗi PLC1 từ AI_PLC1_EStop_Latch
   RUNG wire#powerrail
      Contact( "AI_PLC1_EStop_Latch" )
      S_Coil( "AI_PLC1_Loi_Tong" )
   END_RUNG
   // the same network as SCL:
   IF "AI_PLC1_EStop_Latch" THEN "AI_PLC1_Loi_Tong" := TRUE; END_IF;
END_REGION

REGION Network 77: Tổng hợp lỗi PLC1 từ AI_PLC1_Loi_Dry_Run
   RUNG wire#powerrail
      Contact( "AI_PLC1_Loi_Dry_Run" )
      S_Coil( "AI_PLC1_Loi_Tong" )
   END_RUNG
   // the same network as SCL:
   IF "AI_PLC1_Loi_Dry_Run" THEN "AI_PLC1_Loi_Tong" := TRUE; END_IF;
END_REGION

REGION Network 78: Tổng hợp lỗi PLC1 từ AI_PLC1_Loi_Dosing
   RUNG wire#powerrail
      Contact( "AI_PLC1_Loi_Dosing" )
      S_Coil( "AI_PLC1_Loi_Tong" )
   END_RUNG
   // the same network as SCL:
   IF "AI_PLC1_Loi_Dosing" THEN "AI_PLC1_Loi_Tong" := TRUE; END_IF;
END_REGION

REGION Network 79: Tổng hợp lỗi PLC1 từ AI_PLC1_Loi_Truyen_Thong
   RUNG wire#powerrail
      Contact( "AI_PLC1_Loi_Truyen_Thong" )
      S_Coil( "AI_PLC1_Loi_Tong" )
   END_RUNG
   // the same network as SCL:
   IF "AI_PLC1_Loi_Truyen_Thong" THEN "AI_PLC1_Loi_Tong" := TRUE; END_IF;
END_REGION

REGION Network 80: Tổng hợp lỗi PLC1 từ AI_PLC1_Loi_Setpoint
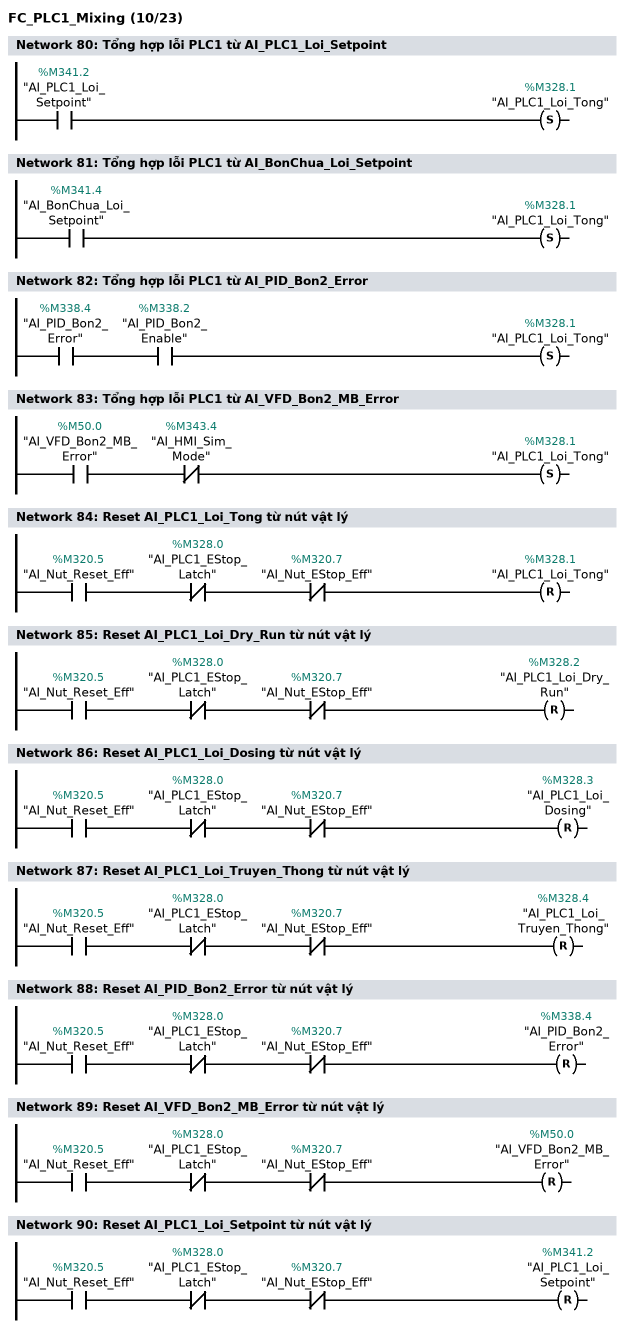
   RUNG wire#powerrail
      Contact( "AI_PLC1_Loi_Setpoint" )
      S_Coil( "AI_PLC1_Loi_Tong" )
   END_RUNG
   // the same network as SCL:
   IF "AI_PLC1_Loi_Setpoint" THEN "AI_PLC1_Loi_Tong" := TRUE; END_IF;
END_REGION

REGION Network 81: Tổng hợp lỗi PLC1 từ AI_BonChua_Loi_Setpoint
   RUNG wire#powerrail
      Contact( "AI_BonChua_Loi_Setpoint" )
      S_Coil( "AI_PLC1_Loi_Tong" )
   END_RUNG
   // the same network as SCL:
   IF "AI_BonChua_Loi_Setpoint" THEN "AI_PLC1_Loi_Tong" := TRUE; END_IF;
END_REGION

REGION Network 82: Tổng hợp lỗi PLC1 từ AI_PID_Bon2_Error
   RUNG wire#powerrail
      Contact( "AI_PID_Bon2_Error" )
      Contact( "AI_PID_Bon2_Enable" )
      S_Coil( "AI_PLC1_Loi_Tong" )
   END_RUNG
   // the same network as SCL:
   IF "AI_PID_Bon2_Error" AND "AI_PID_Bon2_Enable" THEN "AI_PLC1_Loi_Tong" := TRUE; END_IF;
END_REGION

REGION Network 83: Tổng hợp lỗi PLC1 từ AI_VFD_Bon2_MB_Error
   RUNG wire#powerrail
      Contact( "AI_VFD_Bon2_MB_Error" )
      I_Contact( "AI_HMI_Sim_Mode" )
      S_Coil( "AI_PLC1_Loi_Tong" )
   END_RUNG
   // the same network as SCL:
   IF "AI_VFD_Bon2_MB_Error" AND NOT "AI_HMI_Sim_Mode" THEN "AI_PLC1_Loi_Tong" := TRUE; END_IF;
END_REGION

REGION Network 84: Reset AI_PLC1_Loi_Tong từ nút vật lý
   RUNG wire#powerrail
      Contact( "AI_Nut_Reset_Eff" )
      I_Contact( "AI_PLC1_EStop_Latch" )
      I_Contact( "AI_Nut_EStop_Eff" )
      R_Coil( "AI_PLC1_Loi_Tong" )
   END_RUNG
   // the same network as SCL:
   IF "AI_Nut_Reset_Eff" AND NOT "AI_PLC1_EStop_Latch" AND NOT "AI_Nut_EStop_Eff" THEN
       "AI_PLC1_Loi_Tong" := FALSE;
   END_IF;
END_REGION

REGION Network 85: Reset AI_PLC1_Loi_Dry_Run từ nút vật lý
   RUNG wire#powerrail
      Contact( "AI_Nut_Reset_Eff" )
      I_Contact( "AI_PLC1_EStop_Latch" )
      I_Contact( "AI_Nut_EStop_Eff" )
      R_Coil( "AI_PLC1_Loi_Dry_Run" )
   END_RUNG
   // the same network as SCL:
   IF "AI_Nut_Reset_Eff" AND NOT "AI_PLC1_EStop_Latch" AND NOT "AI_Nut_EStop_Eff" THEN
       "AI_PLC1_Loi_Dry_Run" := FALSE;
   END_IF;
END_REGION

REGION Network 86: Reset AI_PLC1_Loi_Dosing từ nút vật lý
   RUNG wire#powerrail
      Contact( "AI_Nut_Reset_Eff" )
      I_Contact( "AI_PLC1_EStop_Latch" )
      I_Contact( "AI_Nut_EStop_Eff" )
      R_Coil( "AI_PLC1_Loi_Dosing" )
   END_RUNG
   // the same network as SCL:
   IF "AI_Nut_Reset_Eff" AND NOT "AI_PLC1_EStop_Latch" AND NOT "AI_Nut_EStop_Eff" THEN
       "AI_PLC1_Loi_Dosing" := FALSE;
   END_IF;
END_REGION

REGION Network 87: Reset AI_PLC1_Loi_Truyen_Thong từ nút vật lý
   RUNG wire#powerrail
      Contact( "AI_Nut_Reset_Eff" )
      I_Contact( "AI_PLC1_EStop_Latch" )
      I_Contact( "AI_Nut_EStop_Eff" )
      R_Coil( "AI_PLC1_Loi_Truyen_Thong" )
   END_RUNG
   // the same network as SCL:
   IF "AI_Nut_Reset_Eff" AND NOT "AI_PLC1_EStop_Latch" AND NOT "AI_Nut_EStop_Eff" THEN
       "AI_PLC1_Loi_Truyen_Thong" := FALSE;
   END_IF;
END_REGION

REGION Network 88: Reset AI_PID_Bon2_Error từ nút vật lý
   RUNG wire#powerrail
      Contact( "AI_Nut_Reset_Eff" )
      I_Contact( "AI_PLC1_EStop_Latch" )
      I_Contact( "AI_Nut_EStop_Eff" )
      R_Coil( "AI_PID_Bon2_Error" )
   END_RUNG
   // the same network as SCL:
   IF "AI_Nut_Reset_Eff" AND NOT "AI_PLC1_EStop_Latch" AND NOT "AI_Nut_EStop_Eff" THEN
       "AI_PID_Bon2_Error" := FALSE;
   END_IF;
END_REGION

REGION Network 89: Reset AI_VFD_Bon2_MB_Error từ nút vật lý
   RUNG wire#powerrail
      Contact( "AI_Nut_Reset_Eff" )
      I_Contact( "AI_PLC1_EStop_Latch" )
      I_Contact( "AI_Nut_EStop_Eff" )
      R_Coil( "AI_VFD_Bon2_MB_Error" )
   END_RUNG
   // the same network as SCL:
   IF "AI_Nut_Reset_Eff" AND NOT "AI_PLC1_EStop_Latch" AND NOT "AI_Nut_EStop_Eff" THEN
       "AI_VFD_Bon2_MB_Error" := FALSE;
   END_IF;
END_REGION

REGION Network 90: Reset AI_PLC1_Loi_Setpoint từ nút vật lý
   RUNG wire#powerrail
      Contact( "AI_Nut_Reset_Eff" )
      I_Contact( "AI_PLC1_EStop_Latch" )
      I_Contact( "AI_Nut_EStop_Eff" )
      R_Coil( "AI_PLC1_Loi_Setpoint" )
   END_RUNG
   // the same network as SCL:
   IF "AI_Nut_Reset_Eff" AND NOT "AI_PLC1_EStop_Latch" AND NOT "AI_Nut_EStop_Eff" THEN
       "AI_PLC1_Loi_Setpoint" := FALSE;
   END_IF;
END_REGION

REGION Network 91: Reset AI_BonChua_Loi_Setpoint từ nút vật lý
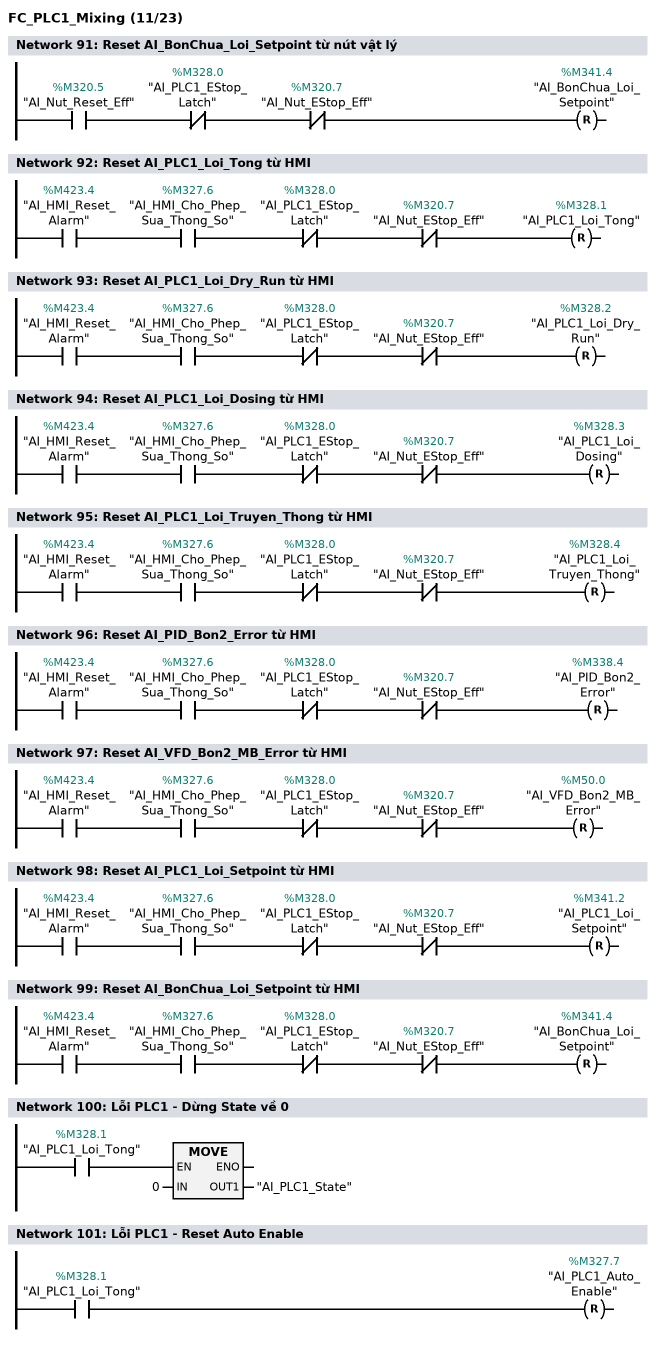
   RUNG wire#powerrail
      Contact( "AI_Nut_Reset_Eff" )
      I_Contact( "AI_PLC1_EStop_Latch" )
      I_Contact( "AI_Nut_EStop_Eff" )
      R_Coil( "AI_BonChua_Loi_Setpoint" )
   END_RUNG
   // the same network as SCL:
   IF "AI_Nut_Reset_Eff" AND NOT "AI_PLC1_EStop_Latch" AND NOT "AI_Nut_EStop_Eff" THEN
       "AI_BonChua_Loi_Setpoint" := FALSE;
   END_IF;
END_REGION

REGION Network 92: Reset AI_PLC1_Loi_Tong từ HMI
   RUNG wire#powerrail
      Contact( "AI_HMI_Reset_Alarm" )
      Contact( "AI_HMI_Cho_Phep_Sua_Thong_So" )
      I_Contact( "AI_PLC1_EStop_Latch" )
      I_Contact( "AI_Nut_EStop_Eff" )
      R_Coil( "AI_PLC1_Loi_Tong" )
   END_RUNG
   // the same network as SCL:
   IF "AI_HMI_Reset_Alarm" AND "AI_HMI_Cho_Phep_Sua_Thong_So" AND NOT "AI_PLC1_EStop_Latch" AND NOT "AI_Nut_EStop_Eff" THEN
       "AI_PLC1_Loi_Tong" := FALSE;
   END_IF;
END_REGION

REGION Network 93: Reset AI_PLC1_Loi_Dry_Run từ HMI
   RUNG wire#powerrail
      Contact( "AI_HMI_Reset_Alarm" )
      Contact( "AI_HMI_Cho_Phep_Sua_Thong_So" )
      I_Contact( "AI_PLC1_EStop_Latch" )
      I_Contact( "AI_Nut_EStop_Eff" )
      R_Coil( "AI_PLC1_Loi_Dry_Run" )
   END_RUNG
   // the same network as SCL:
   IF "AI_HMI_Reset_Alarm" AND "AI_HMI_Cho_Phep_Sua_Thong_So" AND NOT "AI_PLC1_EStop_Latch" AND NOT "AI_Nut_EStop_Eff" THEN
       "AI_PLC1_Loi_Dry_Run" := FALSE;
   END_IF;
END_REGION

REGION Network 94: Reset AI_PLC1_Loi_Dosing từ HMI
   RUNG wire#powerrail
      Contact( "AI_HMI_Reset_Alarm" )
      Contact( "AI_HMI_Cho_Phep_Sua_Thong_So" )
      I_Contact( "AI_PLC1_EStop_Latch" )
      I_Contact( "AI_Nut_EStop_Eff" )
      R_Coil( "AI_PLC1_Loi_Dosing" )
   END_RUNG
   // the same network as SCL:
   IF "AI_HMI_Reset_Alarm" AND "AI_HMI_Cho_Phep_Sua_Thong_So" AND NOT "AI_PLC1_EStop_Latch" AND NOT "AI_Nut_EStop_Eff" THEN
       "AI_PLC1_Loi_Dosing" := FALSE;
   END_IF;
END_REGION

REGION Network 95: Reset AI_PLC1_Loi_Truyen_Thong từ HMI
   RUNG wire#powerrail
      Contact( "AI_HMI_Reset_Alarm" )
      Contact( "AI_HMI_Cho_Phep_Sua_Thong_So" )
      I_Contact( "AI_PLC1_EStop_Latch" )
      I_Contact( "AI_Nut_EStop_Eff" )
      R_Coil( "AI_PLC1_Loi_Truyen_Thong" )
   END_RUNG
   // the same network as SCL:
   IF "AI_HMI_Reset_Alarm" AND "AI_HMI_Cho_Phep_Sua_Thong_So" AND NOT "AI_PLC1_EStop_Latch" AND NOT "AI_Nut_EStop_Eff" THEN
       "AI_PLC1_Loi_Truyen_Thong" := FALSE;
   END_IF;
END_REGION

REGION Network 96: Reset AI_PID_Bon2_Error từ HMI
   RUNG wire#powerrail
      Contact( "AI_HMI_Reset_Alarm" )
      Contact( "AI_HMI_Cho_Phep_Sua_Thong_So" )
      I_Contact( "AI_PLC1_EStop_Latch" )
      I_Contact( "AI_Nut_EStop_Eff" )
      R_Coil( "AI_PID_Bon2_Error" )
   END_RUNG
   // the same network as SCL:
   IF "AI_HMI_Reset_Alarm" AND "AI_HMI_Cho_Phep_Sua_Thong_So" AND NOT "AI_PLC1_EStop_Latch" AND NOT "AI_Nut_EStop_Eff" THEN
       "AI_PID_Bon2_Error" := FALSE;
   END_IF;
END_REGION

REGION Network 97: Reset AI_VFD_Bon2_MB_Error từ HMI
   RUNG wire#powerrail
      Contact( "AI_HMI_Reset_Alarm" )
      Contact( "AI_HMI_Cho_Phep_Sua_Thong_So" )
      I_Contact( "AI_PLC1_EStop_Latch" )
      I_Contact( "AI_Nut_EStop_Eff" )
      R_Coil( "AI_VFD_Bon2_MB_Error" )
   END_RUNG
   // the same network as SCL:
   IF "AI_HMI_Reset_Alarm" AND "AI_HMI_Cho_Phep_Sua_Thong_So" AND NOT "AI_PLC1_EStop_Latch" AND NOT "AI_Nut_EStop_Eff" THEN
       "AI_VFD_Bon2_MB_Error" := FALSE;
   END_IF;
END_REGION

REGION Network 98: Reset AI_PLC1_Loi_Setpoint từ HMI
   RUNG wire#powerrail
      Contact( "AI_HMI_Reset_Alarm" )
      Contact( "AI_HMI_Cho_Phep_Sua_Thong_So" )
      I_Contact( "AI_PLC1_EStop_Latch" )
      I_Contact( "AI_Nut_EStop_Eff" )
      R_Coil( "AI_PLC1_Loi_Setpoint" )
   END_RUNG
   // the same network as SCL:
   IF "AI_HMI_Reset_Alarm" AND "AI_HMI_Cho_Phep_Sua_Thong_So" AND NOT "AI_PLC1_EStop_Latch" AND NOT "AI_Nut_EStop_Eff" THEN
       "AI_PLC1_Loi_Setpoint" := FALSE;
   END_IF;
END_REGION

REGION Network 99: Reset AI_BonChua_Loi_Setpoint từ HMI
   RUNG wire#powerrail
      Contact( "AI_HMI_Reset_Alarm" )
      Contact( "AI_HMI_Cho_Phep_Sua_Thong_So" )
      I_Contact( "AI_PLC1_EStop_Latch" )
      I_Contact( "AI_Nut_EStop_Eff" )
      R_Coil( "AI_BonChua_Loi_Setpoint" )
   END_RUNG
   // the same network as SCL:
   IF "AI_HMI_Reset_Alarm" AND "AI_HMI_Cho_Phep_Sua_Thong_So" AND NOT "AI_PLC1_EStop_Latch" AND NOT "AI_Nut_EStop_Eff" THEN
       "AI_BonChua_Loi_Setpoint" := FALSE;
   END_IF;
END_REGION

REGION Network 100: Lỗi PLC1 - Dừng State về 0
   RUNG wire#powerrail
      Contact( "AI_PLC1_Loi_Tong" )
      { S7_GenerateENO := "TRUE" } Move(in := 0, out1 => "AI_PLC1_State")
   END_RUNG
   // the same network as SCL:
   IF "AI_PLC1_Loi_Tong" THEN "AI_PLC1_State" := 0; END_IF;
END_REGION

REGION Network 101: Lỗi PLC1 - Reset Auto Enable
   RUNG wire#powerrail
      Contact( "AI_PLC1_Loi_Tong" )
      R_Coil( "AI_PLC1_Auto_Enable" )
   END_RUNG
   // the same network as SCL:
   IF "AI_PLC1_Loi_Tong" THEN "AI_PLC1_Auto_Enable" := FALSE; END_IF;
END_REGION

REGION Network 102: Lỗi PLC1 - Reset PID Enable
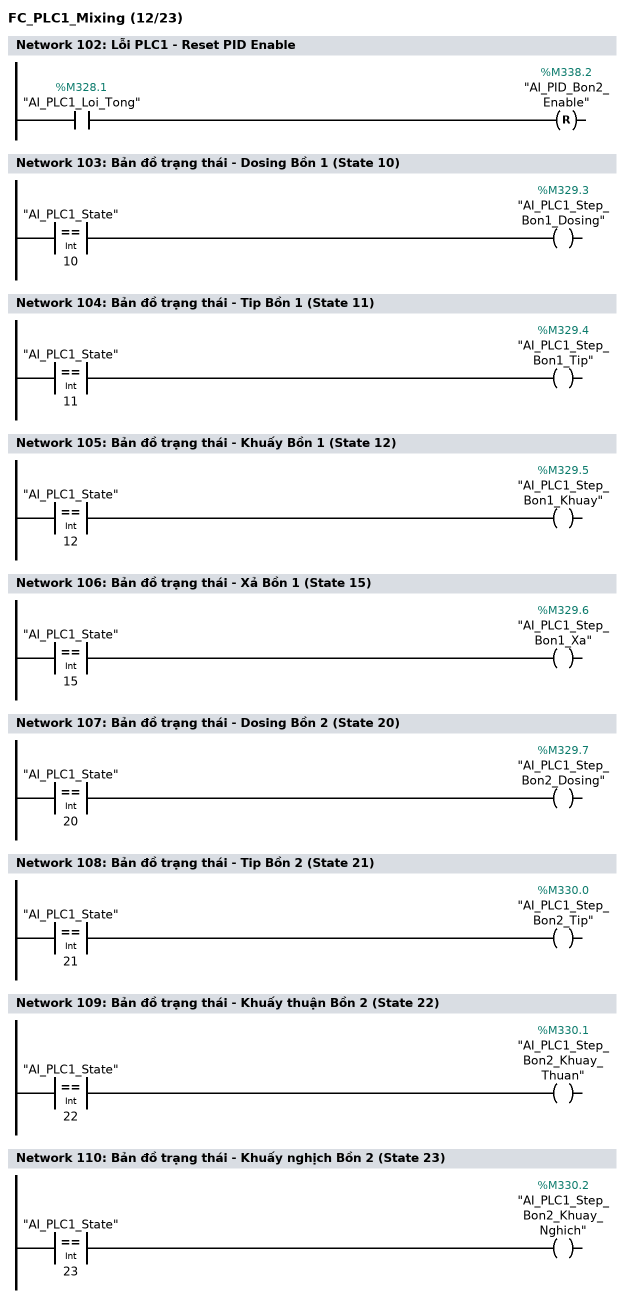
   RUNG wire#powerrail
      Contact( "AI_PLC1_Loi_Tong" )
      R_Coil( "AI_PID_Bon2_Enable" )
   END_RUNG
   // the same network as SCL:
   IF "AI_PLC1_Loi_Tong" THEN "AI_PID_Bon2_Enable" := FALSE; END_IF;
END_REGION

REGION Network 103: Bản đồ trạng thái - Dosing Bồn 1 (State 10)
   RUNG wire#powerrail
      { S7_Templates := "SrcType := Int" } EQ_Contact(in1 := "AI_PLC1_State", in2 := 10)
      Coil( "AI_PLC1_Step_Bon1_Dosing" )
   END_RUNG
   // the same network as SCL:
   "AI_PLC1_Step_Bon1_Dosing" := "AI_PLC1_State" = 10;
END_REGION

REGION Network 104: Bản đồ trạng thái - Tip Bồn 1 (State 11)
   RUNG wire#powerrail
      { S7_Templates := "SrcType := Int" } EQ_Contact(in1 := "AI_PLC1_State", in2 := 11)
      Coil( "AI_PLC1_Step_Bon1_Tip" )
   END_RUNG
   // the same network as SCL:
   "AI_PLC1_Step_Bon1_Tip" := "AI_PLC1_State" = 11;
END_REGION

REGION Network 105: Bản đồ trạng thái - Khuấy Bồn 1 (State 12)
   RUNG wire#powerrail
      { S7_Templates := "SrcType := Int" } EQ_Contact(in1 := "AI_PLC1_State", in2 := 12)
      Coil( "AI_PLC1_Step_Bon1_Khuay" )
   END_RUNG
   // the same network as SCL:
   "AI_PLC1_Step_Bon1_Khuay" := "AI_PLC1_State" = 12;
END_REGION

REGION Network 106: Bản đồ trạng thái - Xả Bồn 1 (State 15)
   RUNG wire#powerrail
      { S7_Templates := "SrcType := Int" } EQ_Contact(in1 := "AI_PLC1_State", in2 := 15)
      Coil( "AI_PLC1_Step_Bon1_Xa" )
   END_RUNG
   // the same network as SCL:
   "AI_PLC1_Step_Bon1_Xa" := "AI_PLC1_State" = 15;
END_REGION

REGION Network 107: Bản đồ trạng thái - Dosing Bồn 2 (State 20)
   RUNG wire#powerrail
      { S7_Templates := "SrcType := Int" } EQ_Contact(in1 := "AI_PLC1_State", in2 := 20)
      Coil( "AI_PLC1_Step_Bon2_Dosing" )
   END_RUNG
   // the same network as SCL:
   "AI_PLC1_Step_Bon2_Dosing" := "AI_PLC1_State" = 20;
END_REGION

REGION Network 108: Bản đồ trạng thái - Tip Bồn 2 (State 21)
   RUNG wire#powerrail
      { S7_Templates := "SrcType := Int" } EQ_Contact(in1 := "AI_PLC1_State", in2 := 21)
      Coil( "AI_PLC1_Step_Bon2_Tip" )
   END_RUNG
   // the same network as SCL:
   "AI_PLC1_Step_Bon2_Tip" := "AI_PLC1_State" = 21;
END_REGION

REGION Network 109: Bản đồ trạng thái - Khuấy thuận Bồn 2 (State 22)
   RUNG wire#powerrail
      { S7_Templates := "SrcType := Int" } EQ_Contact(in1 := "AI_PLC1_State", in2 := 22)
      Coil( "AI_PLC1_Step_Bon2_Khuay_Thuan" )
   END_RUNG
   // the same network as SCL:
   "AI_PLC1_Step_Bon2_Khuay_Thuan" := "AI_PLC1_State" = 22;
END_REGION

REGION Network 110: Bản đồ trạng thái - Khuấy nghịch Bồn 2 (State 23)
   RUNG wire#powerrail
      { S7_Templates := "SrcType := Int" } EQ_Contact(in1 := "AI_PLC1_State", in2 := 23)
      Coil( "AI_PLC1_Step_Bon2_Khuay_Nghich" )
   END_RUNG
   // the same network as SCL:
   "AI_PLC1_Step_Bon2_Khuay_Nghich" := "AI_PLC1_State" = 23;
END_REGION

REGION Network 111: Bản đồ trạng thái - PID Bồn 2 (State 30)
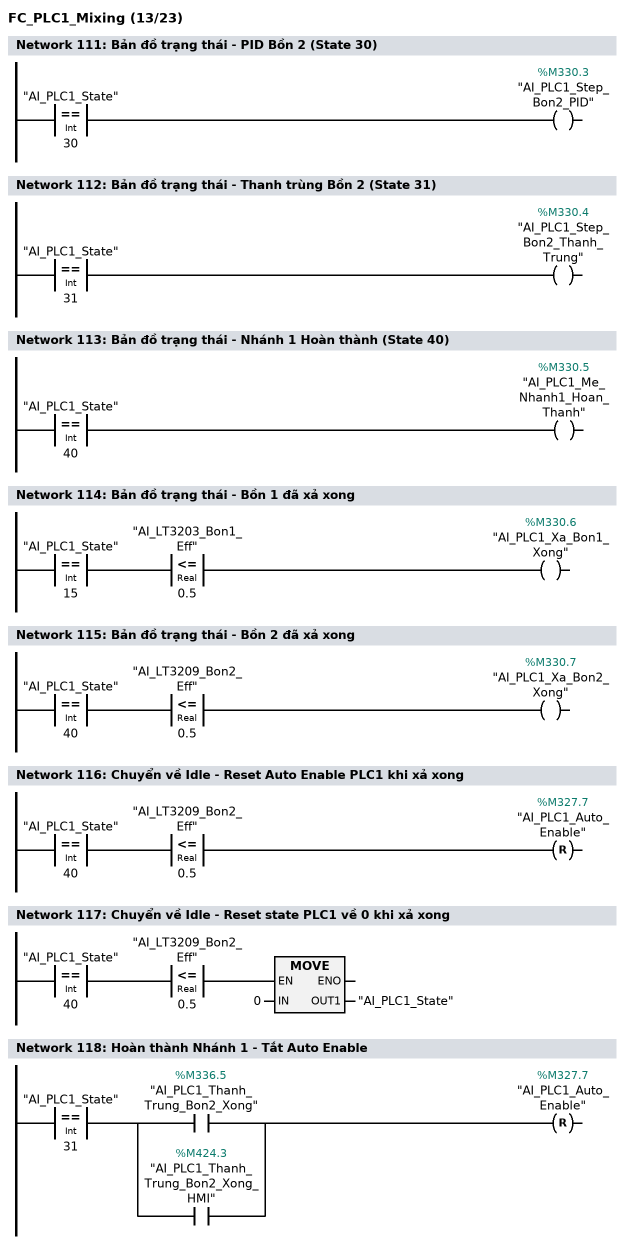
   RUNG wire#powerrail
      { S7_Templates := "SrcType := Int" } EQ_Contact(in1 := "AI_PLC1_State", in2 := 30)
      Coil( "AI_PLC1_Step_Bon2_PID" )
   END_RUNG
   // the same network as SCL:
   "AI_PLC1_Step_Bon2_PID" := "AI_PLC1_State" = 30;
END_REGION

REGION Network 112: Bản đồ trạng thái - Thanh trùng Bồn 2 (State 31)
   RUNG wire#powerrail
      { S7_Templates := "SrcType := Int" } EQ_Contact(in1 := "AI_PLC1_State", in2 := 31)
      Coil( "AI_PLC1_Step_Bon2_Thanh_Trung" )
   END_RUNG
   // the same network as SCL:
   "AI_PLC1_Step_Bon2_Thanh_Trung" := "AI_PLC1_State" = 31;
END_REGION

REGION Network 113: Bản đồ trạng thái - Nhánh 1 Hoàn thành (State 40)
   RUNG wire#powerrail
      { S7_Templates := "SrcType := Int" } EQ_Contact(in1 := "AI_PLC1_State", in2 := 40)
      Coil( "AI_PLC1_Me_Nhanh1_Hoan_Thanh" )
   END_RUNG
   // the same network as SCL:
   "AI_PLC1_Me_Nhanh1_Hoan_Thanh" := "AI_PLC1_State" = 40;
END_REGION

REGION Network 114: Bản đồ trạng thái - Bồn 1 đã xả xong
   RUNG wire#powerrail
      { S7_Templates := "SrcType := Int" } EQ_Contact(in1 := "AI_PLC1_State", in2 := 15)
      { S7_Templates := "SrcType := Real" } LE_Contact(in1 := "AI_LT3203_Bon1_Eff", in2 := 0.5)
      Coil( "AI_PLC1_Xa_Bon1_Xong" )
   END_RUNG
   // the same network as SCL:
   "AI_PLC1_Xa_Bon1_Xong" := ("AI_PLC1_State" = 15) AND ("AI_LT3203_Bon1_Eff" <= 0.5);
END_REGION

REGION Network 115: Bản đồ trạng thái - Bồn 2 đã xả xong
   RUNG wire#powerrail
      { S7_Templates := "SrcType := Int" } EQ_Contact(in1 := "AI_PLC1_State", in2 := 40)
      { S7_Templates := "SrcType := Real" } LE_Contact(in1 := "AI_LT3209_Bon2_Eff", in2 := 0.5)
      Coil( "AI_PLC1_Xa_Bon2_Xong" )
   END_RUNG
   // the same network as SCL:
   "AI_PLC1_Xa_Bon2_Xong" := ("AI_PLC1_State" = 40) AND ("AI_LT3209_Bon2_Eff" <= 0.5);
END_REGION

REGION Network 116: Chuyển về Idle - Reset Auto Enable PLC1 khi xả xong
   RUNG wire#powerrail
      { S7_Templates := "SrcType := Int" } EQ_Contact(in1 := "AI_PLC1_State", in2 := 40)
      { S7_Templates := "SrcType := Real" } LE_Contact(in1 := "AI_LT3209_Bon2_Eff", in2 := 0.5)
      R_Coil( "AI_PLC1_Auto_Enable" )
   END_RUNG
   // the same network as SCL:
   IF ("AI_PLC1_State" = 40) AND ("AI_LT3209_Bon2_Eff" <= 0.5) THEN "AI_PLC1_Auto_Enable" := FALSE; END_IF;
END_REGION

REGION Network 117: Chuyển về Idle - Reset state PLC1 về 0 khi xả xong
   RUNG wire#powerrail
      { S7_Templates := "SrcType := Int" } EQ_Contact(in1 := "AI_PLC1_State", in2 := 40)
      { S7_Templates := "SrcType := Real" } LE_Contact(in1 := "AI_LT3209_Bon2_Eff", in2 := 0.5)
      { S7_GenerateENO := "TRUE" } Move(in := 0, out1 => "AI_PLC1_State")
   END_RUNG
   // the same network as SCL:
   IF ("AI_PLC1_State" = 40) AND ("AI_LT3209_Bon2_Eff" <= 0.5) THEN "AI_PLC1_State" := 0; END_IF;
END_REGION

REGION Network 118: Hoàn thành Nhánh 1 - Tắt Auto Enable
   RUNG wire#powerrail
      { S7_Templates := "SrcType := Int" } EQ_Contact(in1 := "AI_PLC1_State", in2 := 31)
      wire#w1
      Contact( "AI_PLC1_Thanh_Trung_Bon2_Xong" )
      wire#w2
      R_Coil( "AI_PLC1_Auto_Enable" )
   END_RUNG
   RUNG wire#w1
      Contact( "AI_PLC1_Thanh_Trung_Bon2_Xong_HMI" )
   END_RUNG wire#w2
   // the same network as SCL:
   IF ("AI_PLC1_State" = 31) AND ("AI_PLC1_Thanh_Trung_Bon2_Xong" OR "AI_PLC1_Thanh_Trung_Bon2_Xong_HMI") THEN
       "AI_PLC1_Auto_Enable" := FALSE;
   END_IF;
END_REGION

REGION Network 119: Hoàn thành Nhánh 1 - Tắt PID Enable
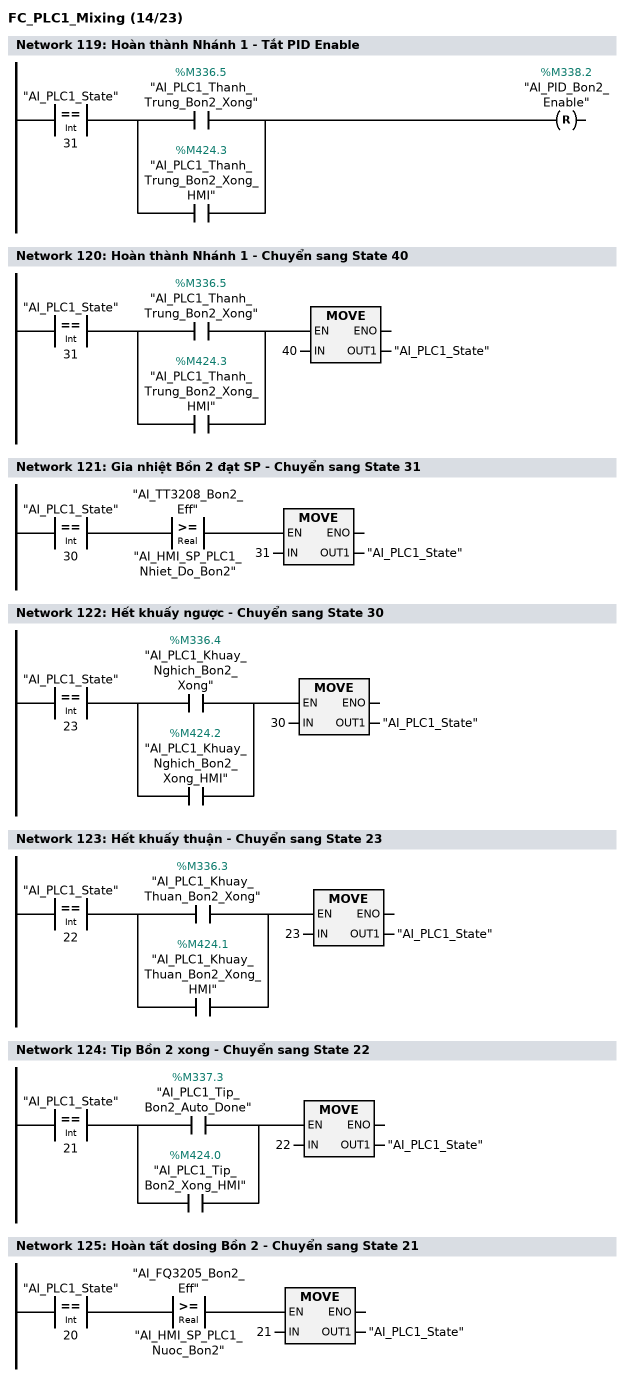
   RUNG wire#powerrail
      { S7_Templates := "SrcType := Int" } EQ_Contact(in1 := "AI_PLC1_State", in2 := 31)
      wire#w1
      Contact( "AI_PLC1_Thanh_Trung_Bon2_Xong" )
      wire#w2
      R_Coil( "AI_PID_Bon2_Enable" )
   END_RUNG
   RUNG wire#w1
      Contact( "AI_PLC1_Thanh_Trung_Bon2_Xong_HMI" )
   END_RUNG wire#w2
   // the same network as SCL:
   IF ("AI_PLC1_State" = 31) AND ("AI_PLC1_Thanh_Trung_Bon2_Xong" OR "AI_PLC1_Thanh_Trung_Bon2_Xong_HMI") THEN
       "AI_PID_Bon2_Enable" := FALSE;
   END_IF;
END_REGION

REGION Network 120: Hoàn thành Nhánh 1 - Chuyển sang State 40
   RUNG wire#powerrail
      { S7_Templates := "SrcType := Int" } EQ_Contact(in1 := "AI_PLC1_State", in2 := 31)
      wire#w1
      Contact( "AI_PLC1_Thanh_Trung_Bon2_Xong" )
      wire#w2
      { S7_GenerateENO := "TRUE" } Move(in := 40, out1 => "AI_PLC1_State")
   END_RUNG
   RUNG wire#w1
      Contact( "AI_PLC1_Thanh_Trung_Bon2_Xong_HMI" )
   END_RUNG wire#w2
   // the same network as SCL:
   IF ("AI_PLC1_State" = 31) AND ("AI_PLC1_Thanh_Trung_Bon2_Xong" OR "AI_PLC1_Thanh_Trung_Bon2_Xong_HMI") THEN
       "AI_PLC1_State" := 40;
   END_IF;
END_REGION

REGION Network 121: Gia nhiệt Bồn 2 đạt SP - Chuyển sang State 31
   RUNG wire#powerrail
      { S7_Templates := "SrcType := Int" } EQ_Contact(in1 := "AI_PLC1_State", in2 := 30)
      { S7_Templates := "SrcType := Real" } GE_Contact(in1 := "AI_TT3208_Bon2_Eff", in2 := "AI_HMI_SP_PLC1_Nhiet_Do_Bon2")
      { S7_GenerateENO := "TRUE" } Move(in := 31, out1 => "AI_PLC1_State")
   END_RUNG
   // the same network as SCL:
   IF ("AI_PLC1_State" = 30) AND ("AI_TT3208_Bon2_Eff" >= "AI_HMI_SP_PLC1_Nhiet_Do_Bon2") THEN
       "AI_PLC1_State" := 31;
   END_IF;
END_REGION

REGION Network 122: Hết khuấy ngược - Chuyển sang State 30
   RUNG wire#powerrail
      { S7_Templates := "SrcType := Int" } EQ_Contact(in1 := "AI_PLC1_State", in2 := 23)
      wire#w1
      Contact( "AI_PLC1_Khuay_Nghich_Bon2_Xong" )
      wire#w2
      { S7_GenerateENO := "TRUE" } Move(in := 30, out1 => "AI_PLC1_State")
   END_RUNG
   RUNG wire#w1
      Contact( "AI_PLC1_Khuay_Nghich_Bon2_Xong_HMI" )
   END_RUNG wire#w2
   // the same network as SCL:
   IF ("AI_PLC1_State" = 23) AND ("AI_PLC1_Khuay_Nghich_Bon2_Xong" OR "AI_PLC1_Khuay_Nghich_Bon2_Xong_HMI") THEN
       "AI_PLC1_State" := 30;
   END_IF;
END_REGION

REGION Network 123: Hết khuấy thuận - Chuyển sang State 23
   RUNG wire#powerrail
      { S7_Templates := "SrcType := Int" } EQ_Contact(in1 := "AI_PLC1_State", in2 := 22)
      wire#w1
      Contact( "AI_PLC1_Khuay_Thuan_Bon2_Xong" )
      wire#w2
      { S7_GenerateENO := "TRUE" } Move(in := 23, out1 => "AI_PLC1_State")
   END_RUNG
   RUNG wire#w1
      Contact( "AI_PLC1_Khuay_Thuan_Bon2_Xong_HMI" )
   END_RUNG wire#w2
   // the same network as SCL:
   IF ("AI_PLC1_State" = 22) AND ("AI_PLC1_Khuay_Thuan_Bon2_Xong" OR "AI_PLC1_Khuay_Thuan_Bon2_Xong_HMI") THEN
       "AI_PLC1_State" := 23;
   END_IF;
END_REGION

REGION Network 124: Tip Bồn 2 xong - Chuyển sang State 22
   RUNG wire#powerrail
      { S7_Templates := "SrcType := Int" } EQ_Contact(in1 := "AI_PLC1_State", in2 := 21)
      wire#w1
      Contact( "AI_PLC1_Tip_Bon2_Auto_Done" )
      wire#w2
      { S7_GenerateENO := "TRUE" } Move(in := 22, out1 => "AI_PLC1_State")
   END_RUNG
   RUNG wire#w1
      Contact( "AI_PLC1_Tip_Bon2_Xong_HMI" )
   END_RUNG wire#w2
   // the same network as SCL:
   IF ("AI_PLC1_State" = 21) AND ("AI_PLC1_Tip_Bon2_Auto_Done" OR "AI_PLC1_Tip_Bon2_Xong_HMI") THEN
       "AI_PLC1_State" := 22;
   END_IF;
END_REGION

REGION Network 125: Hoàn tất dosing Bồn 2 - Chuyển sang State 21
   RUNG wire#powerrail
      { S7_Templates := "SrcType := Int" } EQ_Contact(in1 := "AI_PLC1_State", in2 := 20)
      { S7_Templates := "SrcType := Real" } GE_Contact(in1 := "AI_FQ3205_Bon2_Eff", in2 := "AI_HMI_SP_PLC1_Nuoc_Bon2")
      { S7_GenerateENO := "TRUE" } Move(in := 21, out1 => "AI_PLC1_State")
   END_RUNG
   // the same network as SCL:
   IF ("AI_PLC1_State" = 20) AND ("AI_FQ3205_Bon2_Eff" >= "AI_HMI_SP_PLC1_Nuoc_Bon2") THEN
       "AI_PLC1_State" := 21;
   END_IF;
END_REGION

REGION Network 126: Xả Bồn 1 xong - Chuyển sang State 20
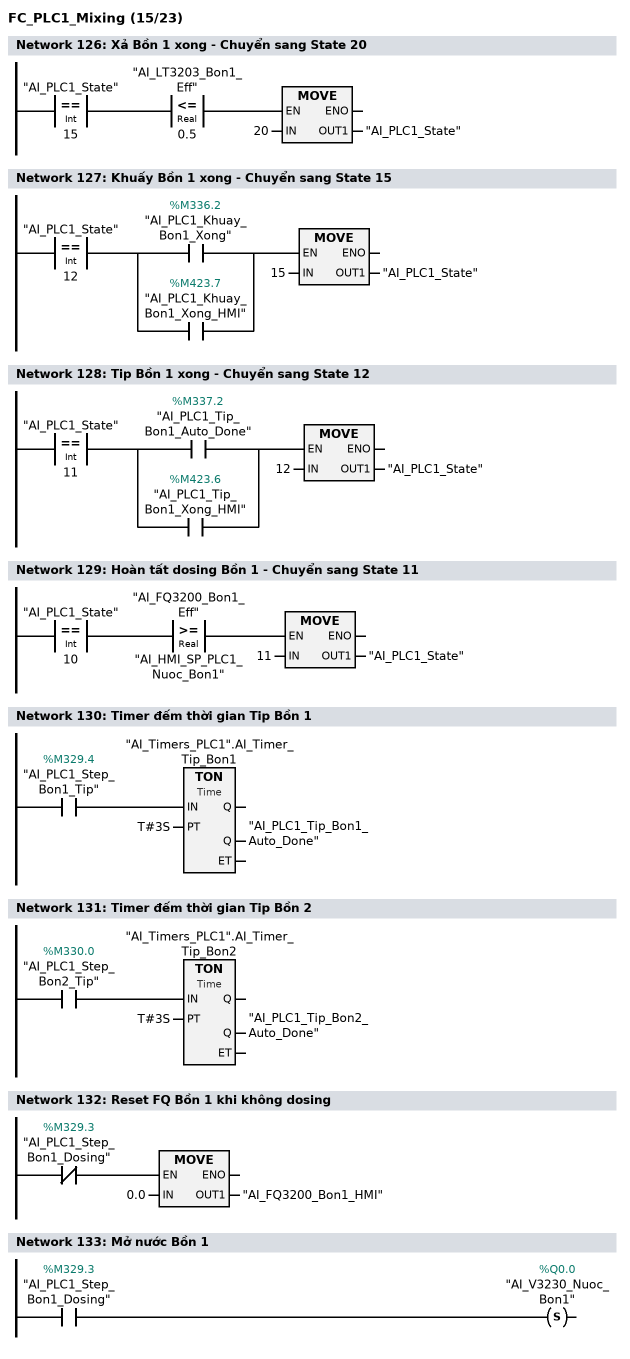
   RUNG wire#powerrail
      { S7_Templates := "SrcType := Int" } EQ_Contact(in1 := "AI_PLC1_State", in2 := 15)
      { S7_Templates := "SrcType := Real" } LE_Contact(in1 := "AI_LT3203_Bon1_Eff", in2 := 0.5)
      { S7_GenerateENO := "TRUE" } Move(in := 20, out1 => "AI_PLC1_State")
   END_RUNG
   // the same network as SCL:
   IF ("AI_PLC1_State" = 15) AND ("AI_LT3203_Bon1_Eff" <= 0.5) THEN "AI_PLC1_State" := 20; END_IF;
END_REGION

REGION Network 127: Khuấy Bồn 1 xong - Chuyển sang State 15
   RUNG wire#powerrail
      { S7_Templates := "SrcType := Int" } EQ_Contact(in1 := "AI_PLC1_State", in2 := 12)
      wire#w1
      Contact( "AI_PLC1_Khuay_Bon1_Xong" )
      wire#w2
      { S7_GenerateENO := "TRUE" } Move(in := 15, out1 => "AI_PLC1_State")
   END_RUNG
   RUNG wire#w1
      Contact( "AI_PLC1_Khuay_Bon1_Xong_HMI" )
   END_RUNG wire#w2
   // the same network as SCL:
   IF ("AI_PLC1_State" = 12) AND ("AI_PLC1_Khuay_Bon1_Xong" OR "AI_PLC1_Khuay_Bon1_Xong_HMI") THEN
       "AI_PLC1_State" := 15;
   END_IF;
END_REGION

REGION Network 128: Tip Bồn 1 xong - Chuyển sang State 12
   RUNG wire#powerrail
      { S7_Templates := "SrcType := Int" } EQ_Contact(in1 := "AI_PLC1_State", in2 := 11)
      wire#w1
      Contact( "AI_PLC1_Tip_Bon1_Auto_Done" )
      wire#w2
      { S7_GenerateENO := "TRUE" } Move(in := 12, out1 => "AI_PLC1_State")
   END_RUNG
   RUNG wire#w1
      Contact( "AI_PLC1_Tip_Bon1_Xong_HMI" )
   END_RUNG wire#w2
   // the same network as SCL:
   IF ("AI_PLC1_State" = 11) AND ("AI_PLC1_Tip_Bon1_Auto_Done" OR "AI_PLC1_Tip_Bon1_Xong_HMI") THEN
       "AI_PLC1_State" := 12;
   END_IF;
END_REGION

REGION Network 129: Hoàn tất dosing Bồn 1 - Chuyển sang State 11
   RUNG wire#powerrail
      { S7_Templates := "SrcType := Int" } EQ_Contact(in1 := "AI_PLC1_State", in2 := 10)
      { S7_Templates := "SrcType := Real" } GE_Contact(in1 := "AI_FQ3200_Bon1_Eff", in2 := "AI_HMI_SP_PLC1_Nuoc_Bon1")
      { S7_GenerateENO := "TRUE" } Move(in := 11, out1 => "AI_PLC1_State")
   END_RUNG
   // the same network as SCL:
   IF ("AI_PLC1_State" = 10) AND ("AI_FQ3200_Bon1_Eff" >= "AI_HMI_SP_PLC1_Nuoc_Bon1") THEN
       "AI_PLC1_State" := 11;
   END_IF;
END_REGION

REGION Network 130: Timer đếm thời gian Tip Bồn 1
   RUNG wire#powerrail
      Contact( "AI_PLC1_Step_Bon1_Tip" )
      { S7_Templates := "time_type := Time" } "AI_Timers_PLC1".AI_Timer_Tip_Bon1.TON(pt := T#3S, q => "AI_PLC1_Tip_Bon1_Auto_Done", et =>)
   END_RUNG
   // the same network as SCL:
   "AI_Timers_PLC1".AI_Timer_Tip_Bon1.TON(IN := "AI_PLC1_Step_Bon1_Tip",
                           PT := T#3S,
                           Q => "AI_PLC1_Tip_Bon1_Auto_Done");
END_REGION

REGION Network 131: Timer đếm thời gian Tip Bồn 2
   RUNG wire#powerrail
      Contact( "AI_PLC1_Step_Bon2_Tip" )
      { S7_Templates := "time_type := Time" } "AI_Timers_PLC1".AI_Timer_Tip_Bon2.TON(pt := T#3S, q => "AI_PLC1_Tip_Bon2_Auto_Done", et =>)
   END_RUNG
   // the same network as SCL:
   "AI_Timers_PLC1".AI_Timer_Tip_Bon2.TON(IN := "AI_PLC1_Step_Bon2_Tip",
                           PT := T#3S,
                           Q => "AI_PLC1_Tip_Bon2_Auto_Done");
END_REGION

REGION Network 132: Reset FQ Bồn 1 khi không dosing
   RUNG wire#powerrail
      I_Contact( "AI_PLC1_Step_Bon1_Dosing" )
      { S7_GenerateENO := "TRUE" } Move(in := 0.0, out1 => "AI_FQ3200_Bon1_HMI")
   END_RUNG
   // the same network as SCL:
   IF NOT "AI_PLC1_Step_Bon1_Dosing" THEN "AI_FQ3200_Bon1_HMI" := 0.0; END_IF;
END_REGION

REGION Network 133: Mở nước Bồn 1
   RUNG wire#powerrail
      Contact( "AI_PLC1_Step_Bon1_Dosing" )
      S_Coil( "AI_V3230_Nuoc_Bon1" )
   END_RUNG
   // the same network as SCL:
   IF "AI_PLC1_Step_Bon1_Dosing" THEN "AI_V3230_Nuoc_Bon1" := TRUE; END_IF;
END_REGION

REGION Network 134: CV nước Bồn 1 mở 100 phần trăm
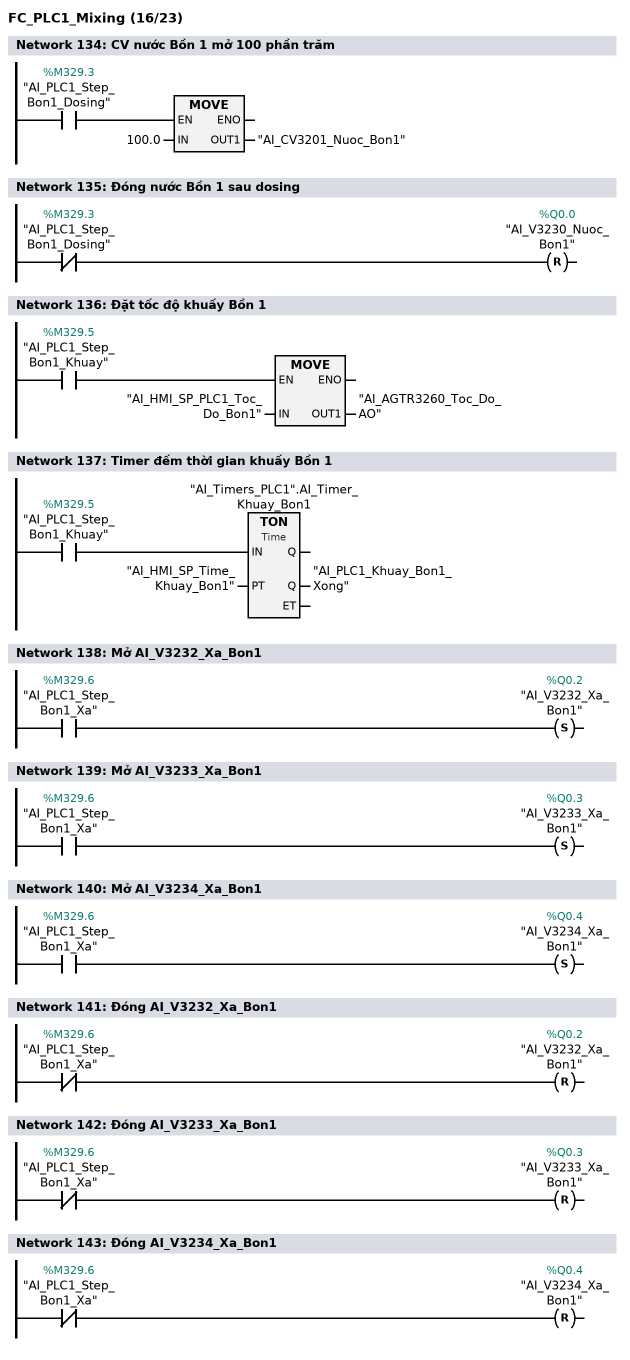
   RUNG wire#powerrail
      Contact( "AI_PLC1_Step_Bon1_Dosing" )
      { S7_GenerateENO := "TRUE" } Move(in := 100.0, out1 => "AI_CV3201_Nuoc_Bon1")
   END_RUNG
   // the same network as SCL:
   IF "AI_PLC1_Step_Bon1_Dosing" THEN "AI_CV3201_Nuoc_Bon1" := 100.0; END_IF;
END_REGION

REGION Network 135: Đóng nước Bồn 1 sau dosing
   RUNG wire#powerrail
      I_Contact( "AI_PLC1_Step_Bon1_Dosing" )
      R_Coil( "AI_V3230_Nuoc_Bon1" )
   END_RUNG
   // the same network as SCL:
   IF NOT "AI_PLC1_Step_Bon1_Dosing" THEN "AI_V3230_Nuoc_Bon1" := FALSE; END_IF;
END_REGION

REGION Network 136: Đặt tốc độ khuấy Bồn 1
   RUNG wire#powerrail
      Contact( "AI_PLC1_Step_Bon1_Khuay" )
      { S7_GenerateENO := "TRUE" } Move(in := "AI_HMI_SP_PLC1_Toc_Do_Bon1", out1 => "AI_AGTR3260_Toc_Do_AO")
   END_RUNG
   // the same network as SCL:
   IF "AI_PLC1_Step_Bon1_Khuay" THEN "AI_AGTR3260_Toc_Do_AO" := "AI_HMI_SP_PLC1_Toc_Do_Bon1"; END_IF;
END_REGION

REGION Network 137: Timer đếm thời gian khuấy Bồn 1
   RUNG wire#powerrail
      Contact( "AI_PLC1_Step_Bon1_Khuay" )
      { S7_Templates := "time_type := Time" } "AI_Timers_PLC1".AI_Timer_Khuay_Bon1.TON(pt := "AI_HMI_SP_Time_Khuay_Bon1", q => "AI_PLC1_Khuay_Bon1_Xong", et =>)
   END_RUNG
   // the same network as SCL:
   "AI_Timers_PLC1".AI_Timer_Khuay_Bon1.TON(IN := "AI_PLC1_Step_Bon1_Khuay",
                           PT := "AI_HMI_SP_Time_Khuay_Bon1",
                           Q => "AI_PLC1_Khuay_Bon1_Xong");
END_REGION

REGION Network 138: Mở AI_V3232_Xa_Bon1
   RUNG wire#powerrail
      Contact( "AI_PLC1_Step_Bon1_Xa" )
      S_Coil( "AI_V3232_Xa_Bon1" )
   END_RUNG
   // the same network as SCL:
   IF "AI_PLC1_Step_Bon1_Xa" THEN "AI_V3232_Xa_Bon1" := TRUE; END_IF;
END_REGION

REGION Network 139: Mở AI_V3233_Xa_Bon1
   RUNG wire#powerrail
      Contact( "AI_PLC1_Step_Bon1_Xa" )
      S_Coil( "AI_V3233_Xa_Bon1" )
   END_RUNG
   // the same network as SCL:
   IF "AI_PLC1_Step_Bon1_Xa" THEN "AI_V3233_Xa_Bon1" := TRUE; END_IF;
END_REGION

REGION Network 140: Mở AI_V3234_Xa_Bon1
   RUNG wire#powerrail
      Contact( "AI_PLC1_Step_Bon1_Xa" )
      S_Coil( "AI_V3234_Xa_Bon1" )
   END_RUNG
   // the same network as SCL:
   IF "AI_PLC1_Step_Bon1_Xa" THEN "AI_V3234_Xa_Bon1" := TRUE; END_IF;
END_REGION

REGION Network 141: Đóng AI_V3232_Xa_Bon1
   RUNG wire#powerrail
      I_Contact( "AI_PLC1_Step_Bon1_Xa" )
      R_Coil( "AI_V3232_Xa_Bon1" )
   END_RUNG
   // the same network as SCL:
   IF NOT "AI_PLC1_Step_Bon1_Xa" THEN "AI_V3232_Xa_Bon1" := FALSE; END_IF;
END_REGION

REGION Network 142: Đóng AI_V3233_Xa_Bon1
   RUNG wire#powerrail
      I_Contact( "AI_PLC1_Step_Bon1_Xa" )
      R_Coil( "AI_V3233_Xa_Bon1" )
   END_RUNG
   // the same network as SCL:
   IF NOT "AI_PLC1_Step_Bon1_Xa" THEN "AI_V3233_Xa_Bon1" := FALSE; END_IF;
END_REGION

REGION Network 143: Đóng AI_V3234_Xa_Bon1
   RUNG wire#powerrail
      I_Contact( "AI_PLC1_Step_Bon1_Xa" )
      R_Coil( "AI_V3234_Xa_Bon1" )
   END_RUNG
   // the same network as SCL:
   IF NOT "AI_PLC1_Step_Bon1_Xa" THEN "AI_V3234_Xa_Bon1" := FALSE; END_IF;
END_REGION

REGION Network 144: Reset FQ Bồn 2 khi không dosing
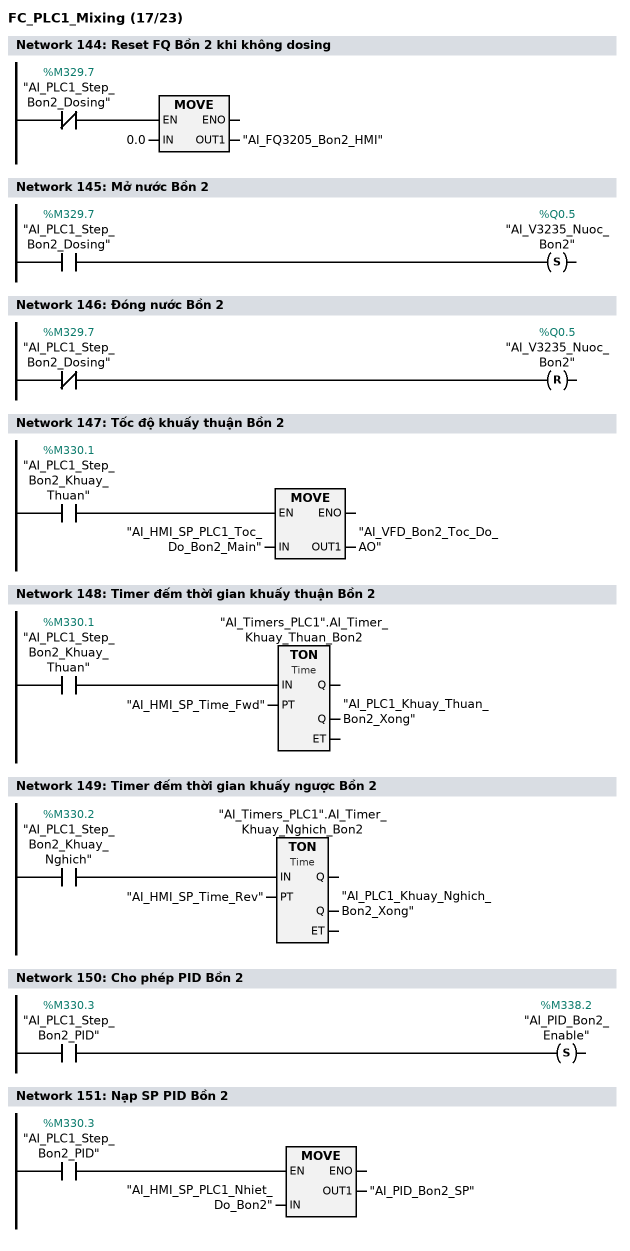
   RUNG wire#powerrail
      I_Contact( "AI_PLC1_Step_Bon2_Dosing" )
      { S7_GenerateENO := "TRUE" } Move(in := 0.0, out1 => "AI_FQ3205_Bon2_HMI")
   END_RUNG
   // the same network as SCL:
   IF NOT "AI_PLC1_Step_Bon2_Dosing" THEN "AI_FQ3205_Bon2_HMI" := 0.0; END_IF;
END_REGION

REGION Network 145: Mở nước Bồn 2
   RUNG wire#powerrail
      Contact( "AI_PLC1_Step_Bon2_Dosing" )
      S_Coil( "AI_V3235_Nuoc_Bon2" )
   END_RUNG
   // the same network as SCL:
   IF "AI_PLC1_Step_Bon2_Dosing" THEN "AI_V3235_Nuoc_Bon2" := TRUE; END_IF;
END_REGION

REGION Network 146: Đóng nước Bồn 2
   RUNG wire#powerrail
      I_Contact( "AI_PLC1_Step_Bon2_Dosing" )
      R_Coil( "AI_V3235_Nuoc_Bon2" )
   END_RUNG
   // the same network as SCL:
   IF NOT "AI_PLC1_Step_Bon2_Dosing" THEN "AI_V3235_Nuoc_Bon2" := FALSE; END_IF;
END_REGION

REGION Network 147: Tốc độ khuấy thuận Bồn 2
   RUNG wire#powerrail
      Contact( "AI_PLC1_Step_Bon2_Khuay_Thuan" )
      { S7_GenerateENO := "TRUE" } Move(in := "AI_HMI_SP_PLC1_Toc_Do_Bon2_Main", out1 => "AI_VFD_Bon2_Toc_Do_AO")
   END_RUNG
   // the same network as SCL:
   IF "AI_PLC1_Step_Bon2_Khuay_Thuan" THEN
       "AI_VFD_Bon2_Toc_Do_AO" := "AI_HMI_SP_PLC1_Toc_Do_Bon2_Main";
   END_IF;
END_REGION

REGION Network 148: Timer đếm thời gian khuấy thuận Bồn 2
   RUNG wire#powerrail
      Contact( "AI_PLC1_Step_Bon2_Khuay_Thuan" )
      { S7_Templates := "time_type := Time" } "AI_Timers_PLC1".AI_Timer_Khuay_Thuan_Bon2.TON(pt := "AI_HMI_SP_Time_Fwd", q => "AI_PLC1_Khuay_Thuan_Bon2_Xong", et =>)
   END_RUNG
   // the same network as SCL:
   "AI_Timers_PLC1".AI_Timer_Khuay_Thuan_Bon2.TON(IN := "AI_PLC1_Step_Bon2_Khuay_Thuan",
                           PT := "AI_HMI_SP_Time_Fwd",
                           Q => "AI_PLC1_Khuay_Thuan_Bon2_Xong");
END_REGION

REGION Network 149: Timer đếm thời gian khuấy ngược Bồn 2
   RUNG wire#powerrail
      Contact( "AI_PLC1_Step_Bon2_Khuay_Nghich" )
      { S7_Templates := "time_type := Time" } "AI_Timers_PLC1".AI_Timer_Khuay_Nghich_Bon2.TON(pt := "AI_HMI_SP_Time_Rev", q => "AI_PLC1_Khuay_Nghich_Bon2_Xong", et =>)
   END_RUNG
   // the same network as SCL:
   "AI_Timers_PLC1".AI_Timer_Khuay_Nghich_Bon2.TON(IN := "AI_PLC1_Step_Bon2_Khuay_Nghich",
                           PT := "AI_HMI_SP_Time_Rev",
                           Q => "AI_PLC1_Khuay_Nghich_Bon2_Xong");
END_REGION

REGION Network 150: Cho phép PID Bồn 2
   RUNG wire#powerrail
      Contact( "AI_PLC1_Step_Bon2_PID" )
      S_Coil( "AI_PID_Bon2_Enable" )
   END_RUNG
   // the same network as SCL:
   IF "AI_PLC1_Step_Bon2_PID" THEN "AI_PID_Bon2_Enable" := TRUE; END_IF;
END_REGION

REGION Network 151: Nạp SP PID Bồn 2
   RUNG wire#powerrail
      Contact( "AI_PLC1_Step_Bon2_PID" )
      { S7_GenerateENO := "TRUE" } Move(in := "AI_HMI_SP_PLC1_Nhiet_Do_Bon2", out1 => "AI_PID_Bon2_SP")
   END_RUNG
   // the same network as SCL:
   IF "AI_PLC1_Step_Bon2_PID" THEN "AI_PID_Bon2_SP" := "AI_HMI_SP_PLC1_Nhiet_Do_Bon2"; END_IF;
END_REGION

REGION Network 152: Timer đếm thời gian thanh trùng Bồn 2
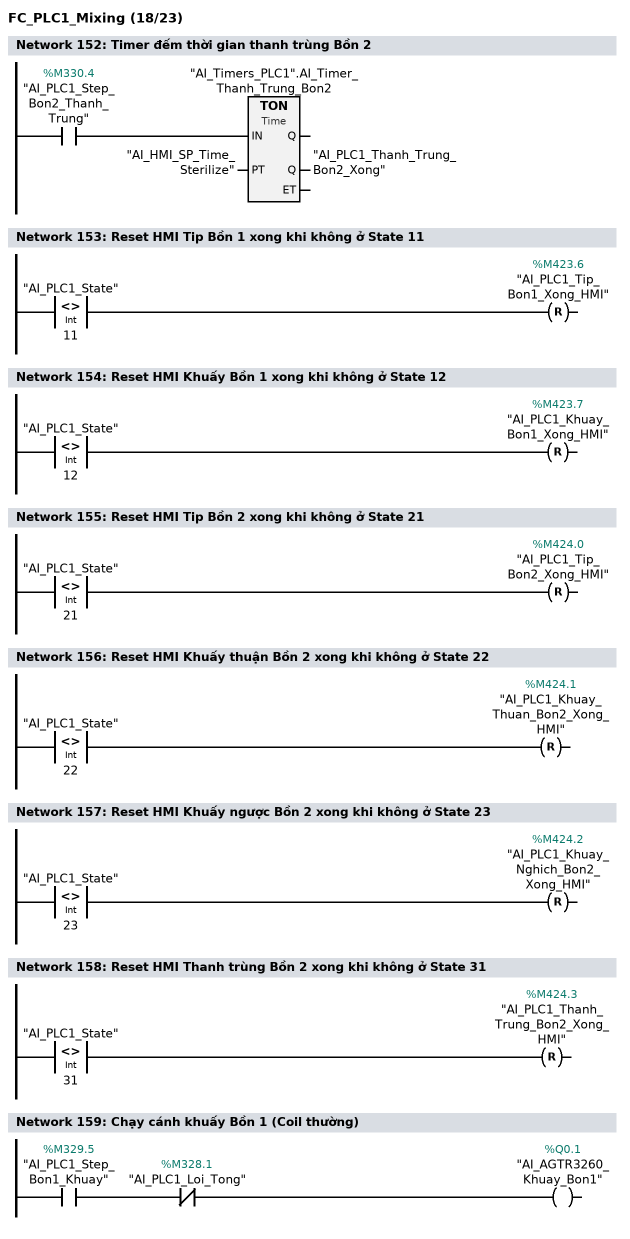
   RUNG wire#powerrail
      Contact( "AI_PLC1_Step_Bon2_Thanh_Trung" )
      { S7_Templates := "time_type := Time" } "AI_Timers_PLC1".AI_Timer_Thanh_Trung_Bon2.TON(pt := "AI_HMI_SP_Time_Sterilize", q => "AI_PLC1_Thanh_Trung_Bon2_Xong", et =>)
   END_RUNG
   // the same network as SCL:
   "AI_Timers_PLC1".AI_Timer_Thanh_Trung_Bon2.TON(IN := "AI_PLC1_Step_Bon2_Thanh_Trung",
                           PT := "AI_HMI_SP_Time_Sterilize",
                           Q => "AI_PLC1_Thanh_Trung_Bon2_Xong");
END_REGION

REGION Network 153: Reset HMI Tip Bồn 1 xong khi không ở State 11
   RUNG wire#powerrail
      { S7_Templates := "SrcType := Int" } NE_Contact(in1 := "AI_PLC1_State", in2 := 11)
      R_Coil( "AI_PLC1_Tip_Bon1_Xong_HMI" )
   END_RUNG
   // the same network as SCL:
   IF "AI_PLC1_State" <> 11 THEN "AI_PLC1_Tip_Bon1_Xong_HMI" := FALSE; END_IF;
END_REGION

REGION Network 154: Reset HMI Khuấy Bồn 1 xong khi không ở State 12
   RUNG wire#powerrail
      { S7_Templates := "SrcType := Int" } NE_Contact(in1 := "AI_PLC1_State", in2 := 12)
      R_Coil( "AI_PLC1_Khuay_Bon1_Xong_HMI" )
   END_RUNG
   // the same network as SCL:
   IF "AI_PLC1_State" <> 12 THEN "AI_PLC1_Khuay_Bon1_Xong_HMI" := FALSE; END_IF;
END_REGION

REGION Network 155: Reset HMI Tip Bồn 2 xong khi không ở State 21
   RUNG wire#powerrail
      { S7_Templates := "SrcType := Int" } NE_Contact(in1 := "AI_PLC1_State", in2 := 21)
      R_Coil( "AI_PLC1_Tip_Bon2_Xong_HMI" )
   END_RUNG
   // the same network as SCL:
   IF "AI_PLC1_State" <> 21 THEN "AI_PLC1_Tip_Bon2_Xong_HMI" := FALSE; END_IF;
END_REGION

REGION Network 156: Reset HMI Khuấy thuận Bồn 2 xong khi không ở State 22
   RUNG wire#powerrail
      { S7_Templates := "SrcType := Int" } NE_Contact(in1 := "AI_PLC1_State", in2 := 22)
      R_Coil( "AI_PLC1_Khuay_Thuan_Bon2_Xong_HMI" )
   END_RUNG
   // the same network as SCL:
   IF "AI_PLC1_State" <> 22 THEN "AI_PLC1_Khuay_Thuan_Bon2_Xong_HMI" := FALSE; END_IF;
END_REGION

REGION Network 157: Reset HMI Khuấy ngược Bồn 2 xong khi không ở State 23
   RUNG wire#powerrail
      { S7_Templates := "SrcType := Int" } NE_Contact(in1 := "AI_PLC1_State", in2 := 23)
      R_Coil( "AI_PLC1_Khuay_Nghich_Bon2_Xong_HMI" )
   END_RUNG
   // the same network as SCL:
   IF "AI_PLC1_State" <> 23 THEN "AI_PLC1_Khuay_Nghich_Bon2_Xong_HMI" := FALSE; END_IF;
END_REGION

REGION Network 158: Reset HMI Thanh trùng Bồn 2 xong khi không ở State 31
   RUNG wire#powerrail
      { S7_Templates := "SrcType := Int" } NE_Contact(in1 := "AI_PLC1_State", in2 := 31)
      R_Coil( "AI_PLC1_Thanh_Trung_Bon2_Xong_HMI" )
   END_RUNG
   // the same network as SCL:
   IF "AI_PLC1_State" <> 31 THEN "AI_PLC1_Thanh_Trung_Bon2_Xong_HMI" := FALSE; END_IF;
END_REGION

REGION Network 159: Chạy cánh khuấy Bồn 1 (Coil thường)
   RUNG wire#powerrail
      Contact( "AI_PLC1_Step_Bon1_Khuay" )
      I_Contact( "AI_PLC1_Loi_Tong" )
      Coil( "AI_AGTR3260_Khuay_Bon1" )
   END_RUNG
   // the same network as SCL:
   "AI_AGTR3260_Khuay_Bon1" := "AI_PLC1_Step_Bon1_Khuay" AND NOT "AI_PLC1_Loi_Tong";
END_REGION

REGION Network 160: Gom trạng thái khuấy thuận/ngược Bồn 2
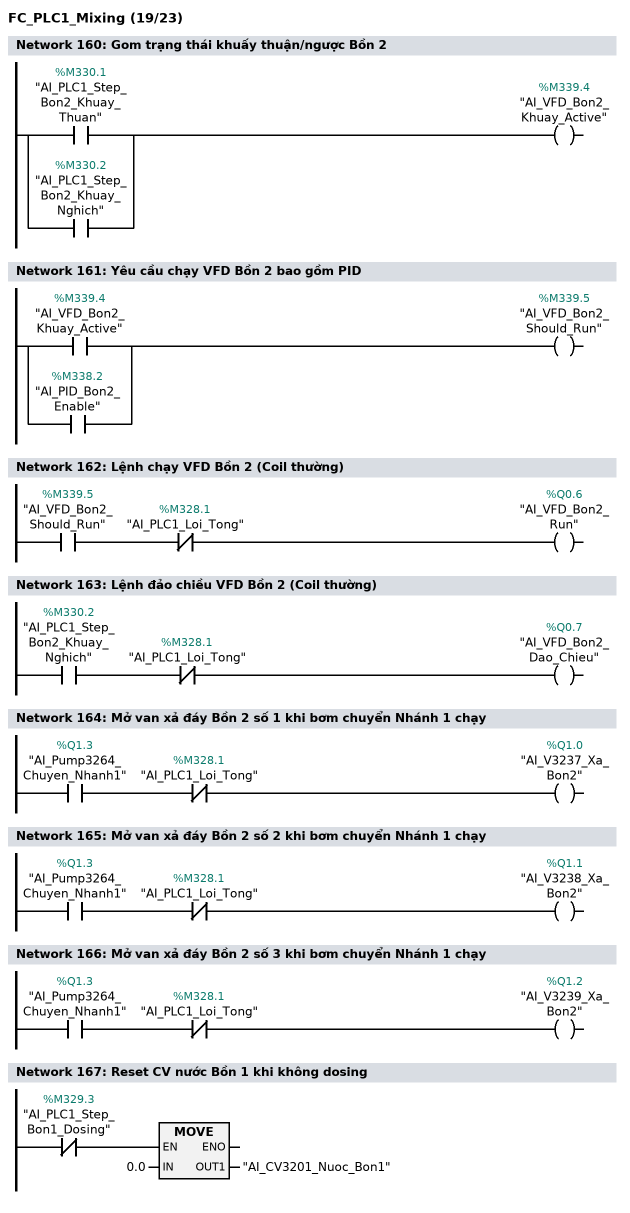
   RUNG wire#powerrail
      Contact( "AI_PLC1_Step_Bon2_Khuay_Thuan" )
      wire#w1
      Coil( "AI_VFD_Bon2_Khuay_Active" )
   END_RUNG
   RUNG wire#powerrail
      Contact( "AI_PLC1_Step_Bon2_Khuay_Nghich" )
   END_RUNG wire#w1
   // the same network as SCL:
   "AI_VFD_Bon2_Khuay_Active" := "AI_PLC1_Step_Bon2_Khuay_Thuan" OR "AI_PLC1_Step_Bon2_Khuay_Nghich";
END_REGION

REGION Network 161: Yêu cầu chạy VFD Bồn 2 bao gồm PID
   RUNG wire#powerrail
      Contact( "AI_VFD_Bon2_Khuay_Active" )
      wire#w1
      Coil( "AI_VFD_Bon2_Should_Run" )
   END_RUNG
   RUNG wire#powerrail
      Contact( "AI_PID_Bon2_Enable" )
   END_RUNG wire#w1
   // the same network as SCL:
   "AI_VFD_Bon2_Should_Run" := "AI_VFD_Bon2_Khuay_Active" OR "AI_PID_Bon2_Enable";
END_REGION

REGION Network 162: Lệnh chạy VFD Bồn 2 (Coil thường)
   RUNG wire#powerrail
      Contact( "AI_VFD_Bon2_Should_Run" )
      I_Contact( "AI_PLC1_Loi_Tong" )
      Coil( "AI_VFD_Bon2_Run" )
   END_RUNG
   // the same network as SCL:
   "AI_VFD_Bon2_Run" := "AI_VFD_Bon2_Should_Run" AND NOT "AI_PLC1_Loi_Tong";
END_REGION

REGION Network 163: Lệnh đảo chiều VFD Bồn 2 (Coil thường)
   RUNG wire#powerrail
      Contact( "AI_PLC1_Step_Bon2_Khuay_Nghich" )
      I_Contact( "AI_PLC1_Loi_Tong" )
      Coil( "AI_VFD_Bon2_Dao_Chieu" )
   END_RUNG
   // the same network as SCL:
   "AI_VFD_Bon2_Dao_Chieu" := "AI_PLC1_Step_Bon2_Khuay_Nghich" AND NOT "AI_PLC1_Loi_Tong";
END_REGION

REGION Network 164: Mở van xả đáy Bồn 2 số 1 khi bơm chuyển Nhánh 1 chạy
   RUNG wire#powerrail
      Contact( "AI_Pump3264_Chuyen_Nhanh1" )
      I_Contact( "AI_PLC1_Loi_Tong" )
      Coil( "AI_V3237_Xa_Bon2" )
   END_RUNG
   // the same network as SCL:
   "AI_V3237_Xa_Bon2" := "AI_Pump3264_Chuyen_Nhanh1" AND NOT "AI_PLC1_Loi_Tong";
END_REGION

REGION Network 165: Mở van xả đáy Bồn 2 số 2 khi bơm chuyển Nhánh 1 chạy
   RUNG wire#powerrail
      Contact( "AI_Pump3264_Chuyen_Nhanh1" )
      I_Contact( "AI_PLC1_Loi_Tong" )
      Coil( "AI_V3238_Xa_Bon2" )
   END_RUNG
   // the same network as SCL:
   "AI_V3238_Xa_Bon2" := "AI_Pump3264_Chuyen_Nhanh1" AND NOT "AI_PLC1_Loi_Tong";
END_REGION

REGION Network 166: Mở van xả đáy Bồn 2 số 3 khi bơm chuyển Nhánh 1 chạy
   RUNG wire#powerrail
      Contact( "AI_Pump3264_Chuyen_Nhanh1" )
      I_Contact( "AI_PLC1_Loi_Tong" )
      Coil( "AI_V3239_Xa_Bon2" )
   END_RUNG
   // the same network as SCL:
   "AI_V3239_Xa_Bon2" := "AI_Pump3264_Chuyen_Nhanh1" AND NOT "AI_PLC1_Loi_Tong";
END_REGION

REGION Network 167: Reset CV nước Bồn 1 khi không dosing
   RUNG wire#powerrail
      I_Contact( "AI_PLC1_Step_Bon1_Dosing" )
      { S7_GenerateENO := "TRUE" } Move(in := 0.0, out1 => "AI_CV3201_Nuoc_Bon1")
   END_RUNG
   // the same network as SCL:
   IF NOT "AI_PLC1_Step_Bon1_Dosing" THEN "AI_CV3201_Nuoc_Bon1" := 0.0; END_IF;
END_REGION

REGION Network 168: Reset CV nước Bồn 1 khi Stop hoặc Lỗi tổng PLC1
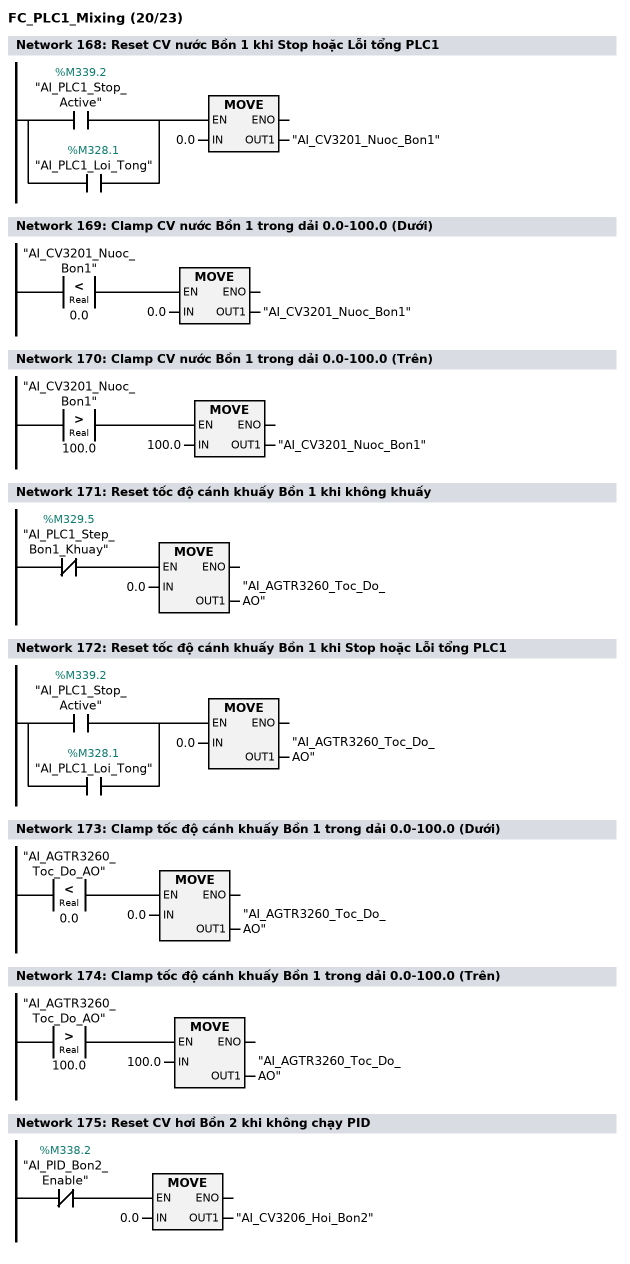
   RUNG wire#powerrail
      Contact( "AI_PLC1_Stop_Active" )
      wire#w1
      { S7_GenerateENO := "TRUE" } Move(in := 0.0, out1 => "AI_CV3201_Nuoc_Bon1")
   END_RUNG
   RUNG wire#powerrail
      Contact( "AI_PLC1_Loi_Tong" )
   END_RUNG wire#w1
   // the same network as SCL:
   IF "AI_PLC1_Stop_Active" OR "AI_PLC1_Loi_Tong" THEN "AI_CV3201_Nuoc_Bon1" := 0.0; END_IF;
END_REGION

REGION Network 169: Clamp CV nước Bồn 1 trong dải 0.0-100.0 (Dưới)
   RUNG wire#powerrail
      { S7_Templates := "SrcType := Real" } LT_Contact(in1 := "AI_CV3201_Nuoc_Bon1", in2 := 0.0)
      { S7_GenerateENO := "TRUE" } Move(in := 0.0, out1 => "AI_CV3201_Nuoc_Bon1")
   END_RUNG
   // the same network as SCL:
   IF "AI_CV3201_Nuoc_Bon1" < 0.0 THEN "AI_CV3201_Nuoc_Bon1" := 0.0; END_IF;
END_REGION

REGION Network 170: Clamp CV nước Bồn 1 trong dải 0.0-100.0 (Trên)
   RUNG wire#powerrail
      { S7_Templates := "SrcType := Real" } GT_Contact(in1 := "AI_CV3201_Nuoc_Bon1", in2 := 100.0)
      { S7_GenerateENO := "TRUE" } Move(in := 100.0, out1 => "AI_CV3201_Nuoc_Bon1")
   END_RUNG
   // the same network as SCL:
   IF "AI_CV3201_Nuoc_Bon1" > 100.0 THEN "AI_CV3201_Nuoc_Bon1" := 100.0; END_IF;
END_REGION

REGION Network 171: Reset tốc độ cánh khuấy Bồn 1 khi không khuấy
   RUNG wire#powerrail
      I_Contact( "AI_PLC1_Step_Bon1_Khuay" )
      { S7_GenerateENO := "TRUE" } Move(in := 0.0, out1 => "AI_AGTR3260_Toc_Do_AO")
   END_RUNG
   // the same network as SCL:
   IF NOT "AI_PLC1_Step_Bon1_Khuay" THEN "AI_AGTR3260_Toc_Do_AO" := 0.0; END_IF;
END_REGION

REGION Network 172: Reset tốc độ cánh khuấy Bồn 1 khi Stop hoặc Lỗi tổng PLC1
   RUNG wire#powerrail
      Contact( "AI_PLC1_Stop_Active" )
      wire#w1
      { S7_GenerateENO := "TRUE" } Move(in := 0.0, out1 => "AI_AGTR3260_Toc_Do_AO")
   END_RUNG
   RUNG wire#powerrail
      Contact( "AI_PLC1_Loi_Tong" )
   END_RUNG wire#w1
   // the same network as SCL:
   IF "AI_PLC1_Stop_Active" OR "AI_PLC1_Loi_Tong" THEN "AI_AGTR3260_Toc_Do_AO" := 0.0; END_IF;
END_REGION

REGION Network 173: Clamp tốc độ cánh khuấy Bồn 1 trong dải 0.0-100.0 (Dưới)
   RUNG wire#powerrail
      { S7_Templates := "SrcType := Real" } LT_Contact(in1 := "AI_AGTR3260_Toc_Do_AO", in2 := 0.0)
      { S7_GenerateENO := "TRUE" } Move(in := 0.0, out1 => "AI_AGTR3260_Toc_Do_AO")
   END_RUNG
   // the same network as SCL:
   IF "AI_AGTR3260_Toc_Do_AO" < 0.0 THEN "AI_AGTR3260_Toc_Do_AO" := 0.0; END_IF;
END_REGION

REGION Network 174: Clamp tốc độ cánh khuấy Bồn 1 trong dải 0.0-100.0 (Trên)
   RUNG wire#powerrail
      { S7_Templates := "SrcType := Real" } GT_Contact(in1 := "AI_AGTR3260_Toc_Do_AO", in2 := 100.0)
      { S7_GenerateENO := "TRUE" } Move(in := 100.0, out1 => "AI_AGTR3260_Toc_Do_AO")
   END_RUNG
   // the same network as SCL:
   IF "AI_AGTR3260_Toc_Do_AO" > 100.0 THEN "AI_AGTR3260_Toc_Do_AO" := 100.0; END_IF;
END_REGION

REGION Network 175: Reset CV hơi Bồn 2 khi không chạy PID
   RUNG wire#powerrail
      I_Contact( "AI_PID_Bon2_Enable" )
      { S7_GenerateENO := "TRUE" } Move(in := 0.0, out1 => "AI_CV3206_Hoi_Bon2")
   END_RUNG
   // the same network as SCL:
   IF NOT "AI_PID_Bon2_Enable" THEN "AI_CV3206_Hoi_Bon2" := 0.0; END_IF;
END_REGION

REGION Network 176: Reset CV hơi Bồn 2 khi Stop hoặc Lỗi tổng PLC1
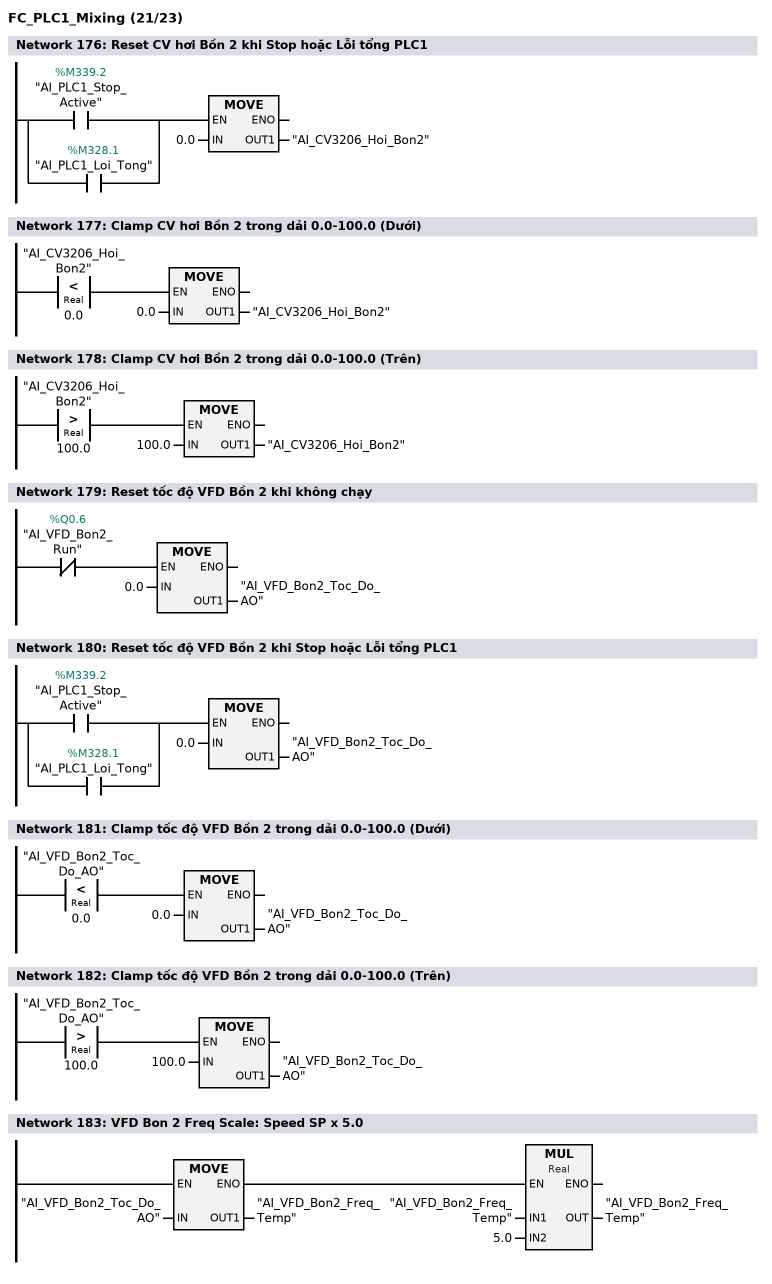
   RUNG wire#powerrail
      Contact( "AI_PLC1_Stop_Active" )
      wire#w1
      { S7_GenerateENO := "TRUE" } Move(in := 0.0, out1 => "AI_CV3206_Hoi_Bon2")
   END_RUNG
   RUNG wire#powerrail
      Contact( "AI_PLC1_Loi_Tong" )
   END_RUNG wire#w1
   // the same network as SCL:
   IF "AI_PLC1_Stop_Active" OR "AI_PLC1_Loi_Tong" THEN "AI_CV3206_Hoi_Bon2" := 0.0; END_IF;
END_REGION

REGION Network 177: Clamp CV hơi Bồn 2 trong dải 0.0-100.0 (Dưới)
   RUNG wire#powerrail
      { S7_Templates := "SrcType := Real" } LT_Contact(in1 := "AI_CV3206_Hoi_Bon2", in2 := 0.0)
      { S7_GenerateENO := "TRUE" } Move(in := 0.0, out1 => "AI_CV3206_Hoi_Bon2")
   END_RUNG
   // the same network as SCL:
   IF "AI_CV3206_Hoi_Bon2" < 0.0 THEN "AI_CV3206_Hoi_Bon2" := 0.0; END_IF;
END_REGION

REGION Network 178: Clamp CV hơi Bồn 2 trong dải 0.0-100.0 (Trên)
   RUNG wire#powerrail
      { S7_Templates := "SrcType := Real" } GT_Contact(in1 := "AI_CV3206_Hoi_Bon2", in2 := 100.0)
      { S7_GenerateENO := "TRUE" } Move(in := 100.0, out1 => "AI_CV3206_Hoi_Bon2")
   END_RUNG
   // the same network as SCL:
   IF "AI_CV3206_Hoi_Bon2" > 100.0 THEN "AI_CV3206_Hoi_Bon2" := 100.0; END_IF;
END_REGION

REGION Network 179: Reset tốc độ VFD Bồn 2 khi không chạy
   RUNG wire#powerrail
      I_Contact( "AI_VFD_Bon2_Run" )
      { S7_GenerateENO := "TRUE" } Move(in := 0.0, out1 => "AI_VFD_Bon2_Toc_Do_AO")
   END_RUNG
   // the same network as SCL:
   IF NOT "AI_VFD_Bon2_Run" THEN "AI_VFD_Bon2_Toc_Do_AO" := 0.0; END_IF;
END_REGION

REGION Network 180: Reset tốc độ VFD Bồn 2 khi Stop hoặc Lỗi tổng PLC1
   RUNG wire#powerrail
      Contact( "AI_PLC1_Stop_Active" )
      wire#w1
      { S7_GenerateENO := "TRUE" } Move(in := 0.0, out1 => "AI_VFD_Bon2_Toc_Do_AO")
   END_RUNG
   RUNG wire#powerrail
      Contact( "AI_PLC1_Loi_Tong" )
   END_RUNG wire#w1
   // the same network as SCL:
   IF "AI_PLC1_Stop_Active" OR "AI_PLC1_Loi_Tong" THEN "AI_VFD_Bon2_Toc_Do_AO" := 0.0; END_IF;
END_REGION

REGION Network 181: Clamp tốc độ VFD Bồn 2 trong dải 0.0-100.0 (Dưới)
   RUNG wire#powerrail
      { S7_Templates := "SrcType := Real" } LT_Contact(in1 := "AI_VFD_Bon2_Toc_Do_AO", in2 := 0.0)
      { S7_GenerateENO := "TRUE" } Move(in := 0.0, out1 => "AI_VFD_Bon2_Toc_Do_AO")
   END_RUNG
   // the same network as SCL:
   IF "AI_VFD_Bon2_Toc_Do_AO" < 0.0 THEN "AI_VFD_Bon2_Toc_Do_AO" := 0.0; END_IF;
END_REGION

REGION Network 182: Clamp tốc độ VFD Bồn 2 trong dải 0.0-100.0 (Trên)
   RUNG wire#powerrail
      { S7_Templates := "SrcType := Real" } GT_Contact(in1 := "AI_VFD_Bon2_Toc_Do_AO", in2 := 100.0)
      { S7_GenerateENO := "TRUE" } Move(in := 100.0, out1 => "AI_VFD_Bon2_Toc_Do_AO")
   END_RUNG
   // the same network as SCL:
   IF "AI_VFD_Bon2_Toc_Do_AO" > 100.0 THEN "AI_VFD_Bon2_Toc_Do_AO" := 100.0; END_IF;
END_REGION

REGION Network 183: VFD Bon 2 Freq Scale: Speed SP x 5.0
   RUNG wire#powerrail
      { S7_GenerateENO := "TRUE" } Move(in := "AI_VFD_Bon2_Toc_Do_AO", out1 => "AI_VFD_Bon2_Freq_Temp")
      { S7_Templates := "SrcType := Real"; S7_GenerateENO := "TRUE" } Mul(in1 := "AI_VFD_Bon2_Freq_Temp", in2 := 5.0, out => "AI_VFD_Bon2_Freq_Temp")
   END_RUNG
   // the same network as SCL:
   // ENO of a box is taken as its EN; it also drops when the box reports an error
   "AI_VFD_Bon2_Freq_Temp" := "AI_VFD_Bon2_Toc_Do_AO";
   "AI_VFD_Bon2_Freq_Temp" := "AI_VFD_Bon2_Freq_Temp" * 5.0;
END_REGION

REGION Network 184: VFD Bon 2 Freq Negate for Reverse Direction
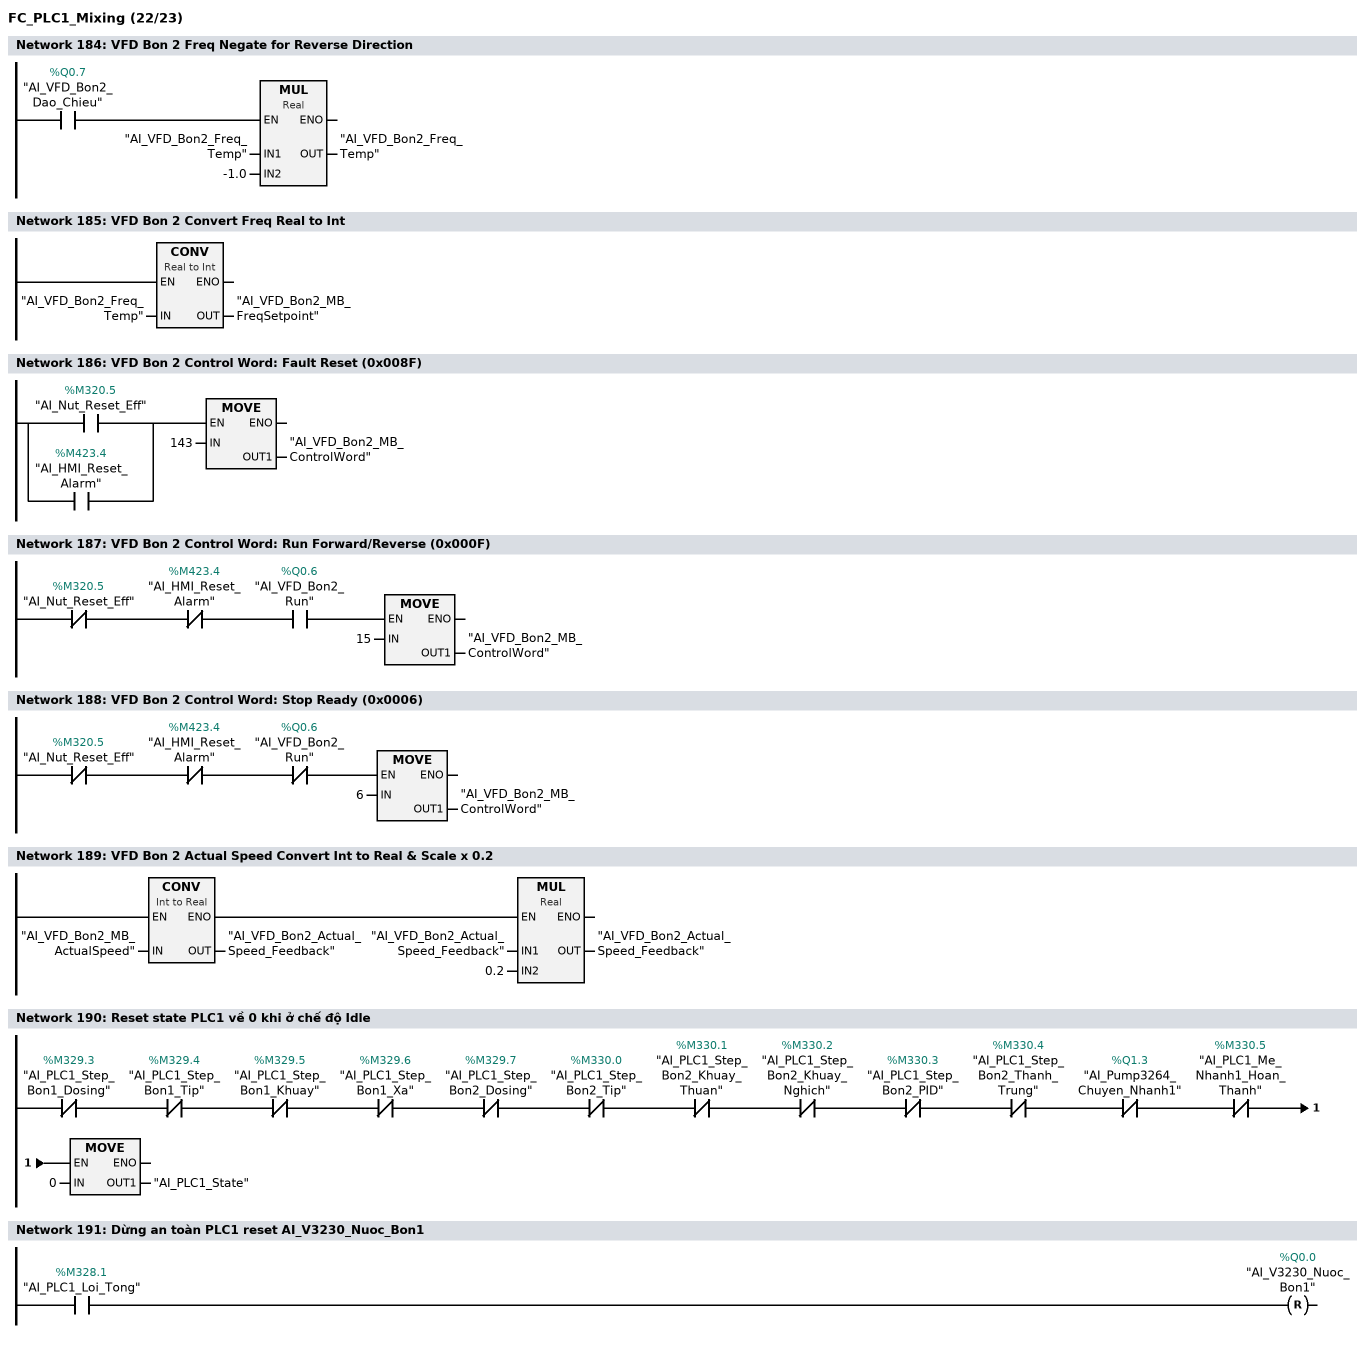
   RUNG wire#powerrail
      Contact( "AI_VFD_Bon2_Dao_Chieu" )
      { S7_Templates := "SrcType := Real"; S7_GenerateENO := "TRUE" } Mul(in1 := "AI_VFD_Bon2_Freq_Temp", in2 := -1.0, out => "AI_VFD_Bon2_Freq_Temp")
   END_RUNG
   // the same network as SCL:
   IF "AI_VFD_Bon2_Dao_Chieu" THEN "AI_VFD_Bon2_Freq_Temp" := "AI_VFD_Bon2_Freq_Temp" * (-1.0); END_IF;
END_REGION

REGION Network 185: VFD Bon 2 Convert Freq Real to Int
   RUNG wire#powerrail
      { S7_Templates := "[SrcType := Real, DestType := Int]"; S7_GenerateENO := "TRUE" } Convert(in := "AI_VFD_Bon2_Freq_Temp", out => "AI_VFD_Bon2_MB_FreqSetpoint")
   END_RUNG
   // the same network as SCL:
   "AI_VFD_Bon2_MB_FreqSetpoint" := REAL_TO_INT("AI_VFD_Bon2_Freq_Temp");
END_REGION

REGION Network 186: VFD Bon 2 Control Word: Fault Reset (0x008F)
   RUNG wire#powerrail
      Contact( "AI_Nut_Reset_Eff" )
      wire#w1
      { S7_GenerateENO := "TRUE" } Move(in := 143, out1 => "AI_VFD_Bon2_MB_ControlWord")
   END_RUNG
   RUNG wire#powerrail
      Contact( "AI_HMI_Reset_Alarm" )
   END_RUNG wire#w1
   // the same network as SCL:
   IF "AI_Nut_Reset_Eff" OR "AI_HMI_Reset_Alarm" THEN "AI_VFD_Bon2_MB_ControlWord" := 143; END_IF;
END_REGION

REGION Network 187: VFD Bon 2 Control Word: Run Forward/Reverse (0x000F)
   RUNG wire#powerrail
      I_Contact( "AI_Nut_Reset_Eff" )
      I_Contact( "AI_HMI_Reset_Alarm" )
      Contact( "AI_VFD_Bon2_Run" )
      { S7_GenerateENO := "TRUE" } Move(in := 15, out1 => "AI_VFD_Bon2_MB_ControlWord")
   END_RUNG
   // the same network as SCL:
   IF NOT "AI_Nut_Reset_Eff" AND NOT "AI_HMI_Reset_Alarm" AND "AI_VFD_Bon2_Run" THEN
       "AI_VFD_Bon2_MB_ControlWord" := 15;
   END_IF;
END_REGION

REGION Network 188: VFD Bon 2 Control Word: Stop Ready (0x0006)
   RUNG wire#powerrail
      I_Contact( "AI_Nut_Reset_Eff" )
      I_Contact( "AI_HMI_Reset_Alarm" )
      I_Contact( "AI_VFD_Bon2_Run" )
      { S7_GenerateENO := "TRUE" } Move(in := 6, out1 => "AI_VFD_Bon2_MB_ControlWord")
   END_RUNG
   // the same network as SCL:
   IF NOT "AI_Nut_Reset_Eff" AND NOT "AI_HMI_Reset_Alarm" AND NOT "AI_VFD_Bon2_Run" THEN
       "AI_VFD_Bon2_MB_ControlWord" := 6;
   END_IF;
END_REGION

REGION Network 189: VFD Bon 2 Actual Speed Convert Int to Real & Scale x 0.2
   RUNG wire#powerrail
      { S7_Templates := "[SrcType := Int, DestType := Real]"; S7_GenerateENO := "TRUE" } Convert(in := "AI_VFD_Bon2_MB_ActualSpeed", out => "AI_VFD_Bon2_Actual_Speed_Feedback")
      { S7_Templates := "SrcType := Real"; S7_GenerateENO := "TRUE" } Mul(in1 := "AI_VFD_Bon2_Actual_Speed_Feedback", in2 := 0.2, out => "AI_VFD_Bon2_Actual_Speed_Feedback")
   END_RUNG
   // the same network as SCL:
   // ENO of a box is taken as its EN; it also drops when the box reports an error
   "AI_VFD_Bon2_Actual_Speed_Feedback" := INT_TO_REAL("AI_VFD_Bon2_MB_ActualSpeed");
   "AI_VFD_Bon2_Actual_Speed_Feedback" := "AI_VFD_Bon2_Actual_Speed_Feedback" * 0.2;
END_REGION

REGION Network 190: Reset state PLC1 về 0 khi ở chế độ Idle
   RUNG wire#powerrail
      I_Contact( "AI_PLC1_Step_Bon1_Dosing" )
      I_Contact( "AI_PLC1_Step_Bon1_Tip" )
      I_Contact( "AI_PLC1_Step_Bon1_Khuay" )
      I_Contact( "AI_PLC1_Step_Bon1_Xa" )
      I_Contact( "AI_PLC1_Step_Bon2_Dosing" )
      I_Contact( "AI_PLC1_Step_Bon2_Tip" )
      I_Contact( "AI_PLC1_Step_Bon2_Khuay_Thuan" )
      I_Contact( "AI_PLC1_Step_Bon2_Khuay_Nghich" )
      I_Contact( "AI_PLC1_Step_Bon2_PID" )
      I_Contact( "AI_PLC1_Step_Bon2_Thanh_Trung" )
      I_Contact( "AI_Pump3264_Chuyen_Nhanh1" )
      I_Contact( "AI_PLC1_Me_Nhanh1_Hoan_Thanh" )
      { S7_GenerateENO := "TRUE" } Move(in := 0, out1 => "AI_PLC1_State")
   END_RUNG
   // the same network as SCL:
   IF NOT "AI_PLC1_Step_Bon1_Dosing" AND NOT "AI_PLC1_Step_Bon1_Tip" AND NOT "AI_PLC1_Step_Bon1_Khuay" AND NOT "AI_PLC1_Step_Bon1_Xa" AND NOT "AI_PLC1_Step_Bon2_Dosing" AND NOT "AI_PLC1_Step_Bon2_Tip" AND NOT "AI_PLC1_Step_Bon2_Khuay_Thuan" AND NOT "AI_PLC1_Step_Bon2_Khuay_Nghich" AND NOT "AI_PLC1_Step_Bon2_PID" AND NOT "AI_PLC1_Step_Bon2_Thanh_Trung" AND NOT "AI_Pump3264_Chuyen_Nhanh1" AND NOT "AI_PLC1_Me_Nhanh1_Hoan_Thanh" THEN
       "AI_PLC1_State" := 0;
   END_IF;
END_REGION

REGION Network 191: Dừng an toàn PLC1 reset AI_V3230_Nuoc_Bon1
   RUNG wire#powerrail
      Contact( "AI_PLC1_Loi_Tong" )
      R_Coil( "AI_V3230_Nuoc_Bon1" )
   END_RUNG
   // the same network as SCL:
   IF "AI_PLC1_Loi_Tong" THEN "AI_V3230_Nuoc_Bon1" := FALSE; END_IF;
END_REGION

REGION Network 192: Dừng an toàn PLC1 reset AI_V3232_Xa_Bon1
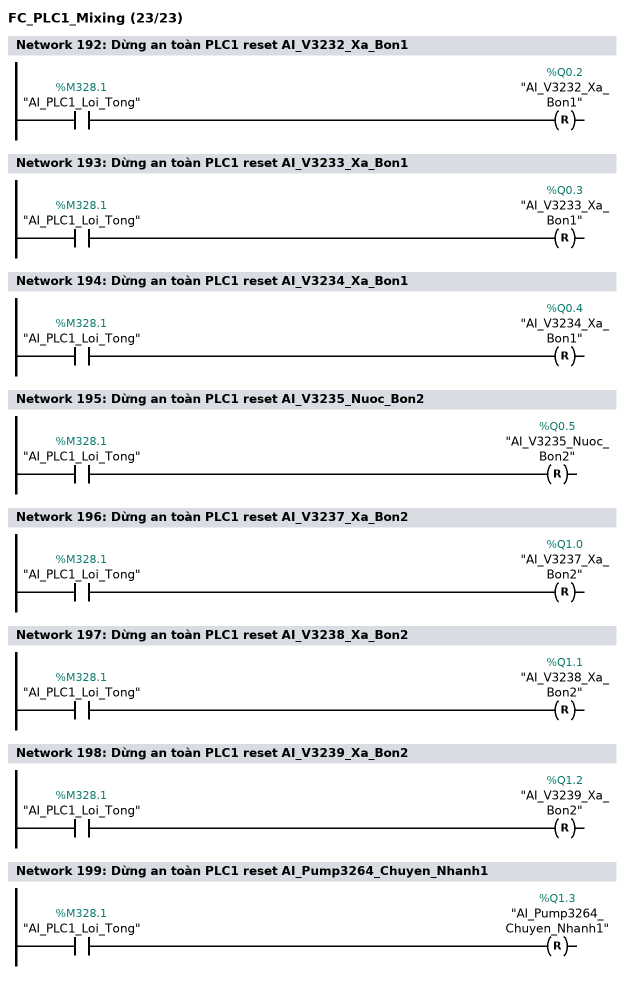
   RUNG wire#powerrail
      Contact( "AI_PLC1_Loi_Tong" )
      R_Coil( "AI_V3232_Xa_Bon1" )
   END_RUNG
   // the same network as SCL:
   IF "AI_PLC1_Loi_Tong" THEN "AI_V3232_Xa_Bon1" := FALSE; END_IF;
END_REGION

REGION Network 193: Dừng an toàn PLC1 reset AI_V3233_Xa_Bon1
   RUNG wire#powerrail
      Contact( "AI_PLC1_Loi_Tong" )
      R_Coil( "AI_V3233_Xa_Bon1" )
   END_RUNG
   // the same network as SCL:
   IF "AI_PLC1_Loi_Tong" THEN "AI_V3233_Xa_Bon1" := FALSE; END_IF;
END_REGION

REGION Network 194: Dừng an toàn PLC1 reset AI_V3234_Xa_Bon1
   RUNG wire#powerrail
      Contact( "AI_PLC1_Loi_Tong" )
      R_Coil( "AI_V3234_Xa_Bon1" )
   END_RUNG
   // the same network as SCL:
   IF "AI_PLC1_Loi_Tong" THEN "AI_V3234_Xa_Bon1" := FALSE; END_IF;
END_REGION

REGION Network 195: Dừng an toàn PLC1 reset AI_V3235_Nuoc_Bon2
   RUNG wire#powerrail
      Contact( "AI_PLC1_Loi_Tong" )
      R_Coil( "AI_V3235_Nuoc_Bon2" )
   END_RUNG
   // the same network as SCL:
   IF "AI_PLC1_Loi_Tong" THEN "AI_V3235_Nuoc_Bon2" := FALSE; END_IF;
END_REGION

REGION Network 196: Dừng an toàn PLC1 reset AI_V3237_Xa_Bon2
   RUNG wire#powerrail
      Contact( "AI_PLC1_Loi_Tong" )
      R_Coil( "AI_V3237_Xa_Bon2" )
   END_RUNG
   // the same network as SCL:
   IF "AI_PLC1_Loi_Tong" THEN "AI_V3237_Xa_Bon2" := FALSE; END_IF;
END_REGION

REGION Network 197: Dừng an toàn PLC1 reset AI_V3238_Xa_Bon2
   RUNG wire#powerrail
      Contact( "AI_PLC1_Loi_Tong" )
      R_Coil( "AI_V3238_Xa_Bon2" )
   END_RUNG
   // the same network as SCL:
   IF "AI_PLC1_Loi_Tong" THEN "AI_V3238_Xa_Bon2" := FALSE; END_IF;
END_REGION

REGION Network 198: Dừng an toàn PLC1 reset AI_V3239_Xa_Bon2
   RUNG wire#powerrail
      Contact( "AI_PLC1_Loi_Tong" )
      R_Coil( "AI_V3239_Xa_Bon2" )
   END_RUNG
   // the same network as SCL:
   IF "AI_PLC1_Loi_Tong" THEN "AI_V3239_Xa_Bon2" := FALSE; END_IF;
END_REGION

REGION Network 199: Dừng an toàn PLC1 reset AI_Pump3264_Chuyen_Nhanh1
   RUNG wire#powerrail
      Contact( "AI_PLC1_Loi_Tong" )
      R_Coil( "AI_Pump3264_Chuyen_Nhanh1" )
   END_RUNG
   // the same network as SCL:
   IF "AI_PLC1_Loi_Tong" THEN "AI_Pump3264_Chuyen_Nhanh1" := FALSE; END_IF;
END_REGION
END_FUNCTION

FUNCTION "FC_HMI_Mirror_PLC2" : Void   // FC41, LAD
{ S7_Optimized_Access := 'TRUE' }
VERSION : 0.1
// stored: AutoNumber true, IsIECCheckEnabled false
BEGIN

REGION Network 1: Mirror AI_V3240_Nuoc_Bon3
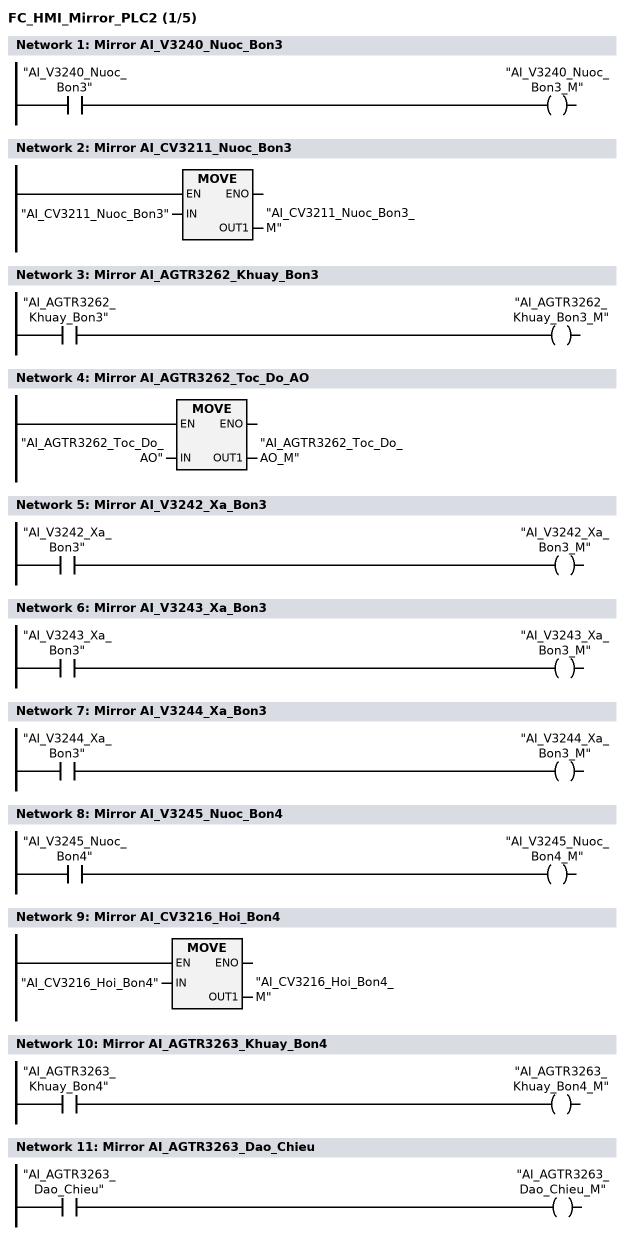
   RUNG wire#powerrail
      Contact( "AI_V3240_Nuoc_Bon3" )
      Coil( "AI_V3240_Nuoc_Bon3_M" )
   END_RUNG
   // the same network as SCL:
   "AI_V3240_Nuoc_Bon3_M" := "AI_V3240_Nuoc_Bon3";
END_REGION

REGION Network 2: Mirror AI_CV3211_Nuoc_Bon3
   RUNG wire#powerrail
      { S7_GenerateENO := "TRUE" } Move(in := "AI_CV3211_Nuoc_Bon3", out1 => "AI_CV3211_Nuoc_Bon3_M")
   END_RUNG
   // the same network as SCL:
   "AI_CV3211_Nuoc_Bon3_M" := "AI_CV3211_Nuoc_Bon3";
END_REGION

REGION Network 3: Mirror AI_AGTR3262_Khuay_Bon3
   RUNG wire#powerrail
      Contact( "AI_AGTR3262_Khuay_Bon3" )
      Coil( "AI_AGTR3262_Khuay_Bon3_M" )
   END_RUNG
   // the same network as SCL:
   "AI_AGTR3262_Khuay_Bon3_M" := "AI_AGTR3262_Khuay_Bon3";
END_REGION

REGION Network 4: Mirror AI_AGTR3262_Toc_Do_AO
   RUNG wire#powerrail
      { S7_GenerateENO := "TRUE" } Move(in := "AI_AGTR3262_Toc_Do_AO", out1 => "AI_AGTR3262_Toc_Do_AO_M")
   END_RUNG
   // the same network as SCL:
   "AI_AGTR3262_Toc_Do_AO_M" := "AI_AGTR3262_Toc_Do_AO";
END_REGION

REGION Network 5: Mirror AI_V3242_Xa_Bon3
   RUNG wire#powerrail
      Contact( "AI_V3242_Xa_Bon3" )
      Coil( "AI_V3242_Xa_Bon3_M" )
   END_RUNG
   // the same network as SCL:
   "AI_V3242_Xa_Bon3_M" := "AI_V3242_Xa_Bon3";
END_REGION

REGION Network 6: Mirror AI_V3243_Xa_Bon3
   RUNG wire#powerrail
      Contact( "AI_V3243_Xa_Bon3" )
      Coil( "AI_V3243_Xa_Bon3_M" )
   END_RUNG
   // the same network as SCL:
   "AI_V3243_Xa_Bon3_M" := "AI_V3243_Xa_Bon3";
END_REGION

REGION Network 7: Mirror AI_V3244_Xa_Bon3
   RUNG wire#powerrail
      Contact( "AI_V3244_Xa_Bon3" )
      Coil( "AI_V3244_Xa_Bon3_M" )
   END_RUNG
   // the same network as SCL:
   "AI_V3244_Xa_Bon3_M" := "AI_V3244_Xa_Bon3";
END_REGION

REGION Network 8: Mirror AI_V3245_Nuoc_Bon4
   RUNG wire#powerrail
      Contact( "AI_V3245_Nuoc_Bon4" )
      Coil( "AI_V3245_Nuoc_Bon4_M" )
   END_RUNG
   // the same network as SCL:
   "AI_V3245_Nuoc_Bon4_M" := "AI_V3245_Nuoc_Bon4";
END_REGION

REGION Network 9: Mirror AI_CV3216_Hoi_Bon4
   RUNG wire#powerrail
      { S7_GenerateENO := "TRUE" } Move(in := "AI_CV3216_Hoi_Bon4", out1 => "AI_CV3216_Hoi_Bon4_M")
   END_RUNG
   // the same network as SCL:
   "AI_CV3216_Hoi_Bon4_M" := "AI_CV3216_Hoi_Bon4";
END_REGION

REGION Network 10: Mirror AI_AGTR3263_Khuay_Bon4
   RUNG wire#powerrail
      Contact( "AI_AGTR3263_Khuay_Bon4" )
      Coil( "AI_AGTR3263_Khuay_Bon4_M" )
   END_RUNG
   // the same network as SCL:
   "AI_AGTR3263_Khuay_Bon4_M" := "AI_AGTR3263_Khuay_Bon4";
END_REGION

REGION Network 11: Mirror AI_AGTR3263_Dao_Chieu
   RUNG wire#powerrail
      Contact( "AI_AGTR3263_Dao_Chieu" )
      Coil( "AI_AGTR3263_Dao_Chieu_M" )
   END_RUNG
   // the same network as SCL:
   "AI_AGTR3263_Dao_Chieu_M" := "AI_AGTR3263_Dao_Chieu";
END_REGION

REGION Network 12: Mirror AI_AGTR3263_Toc_Do_AO
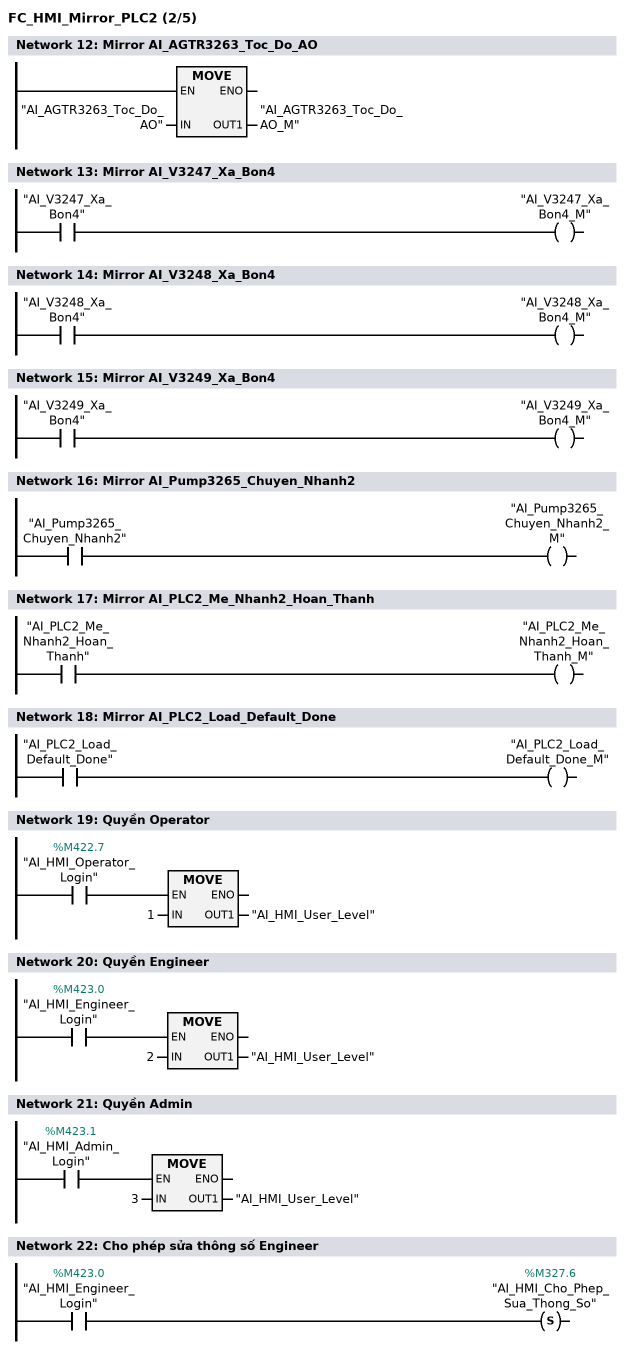
   RUNG wire#powerrail
      { S7_GenerateENO := "TRUE" } Move(in := "AI_AGTR3263_Toc_Do_AO", out1 => "AI_AGTR3263_Toc_Do_AO_M")
   END_RUNG
   // the same network as SCL:
   "AI_AGTR3263_Toc_Do_AO_M" := "AI_AGTR3263_Toc_Do_AO";
END_REGION

REGION Network 13: Mirror AI_V3247_Xa_Bon4
   RUNG wire#powerrail
      Contact( "AI_V3247_Xa_Bon4" )
      Coil( "AI_V3247_Xa_Bon4_M" )
   END_RUNG
   // the same network as SCL:
   "AI_V3247_Xa_Bon4_M" := "AI_V3247_Xa_Bon4";
END_REGION

REGION Network 14: Mirror AI_V3248_Xa_Bon4
   RUNG wire#powerrail
      Contact( "AI_V3248_Xa_Bon4" )
      Coil( "AI_V3248_Xa_Bon4_M" )
   END_RUNG
   // the same network as SCL:
   "AI_V3248_Xa_Bon4_M" := "AI_V3248_Xa_Bon4";
END_REGION

REGION Network 15: Mirror AI_V3249_Xa_Bon4
   RUNG wire#powerrail
      Contact( "AI_V3249_Xa_Bon4" )
      Coil( "AI_V3249_Xa_Bon4_M" )
   END_RUNG
   // the same network as SCL:
   "AI_V3249_Xa_Bon4_M" := "AI_V3249_Xa_Bon4";
END_REGION

REGION Network 16: Mirror AI_Pump3265_Chuyen_Nhanh2
   RUNG wire#powerrail
      Contact( "AI_Pump3265_Chuyen_Nhanh2" )
      Coil( "AI_Pump3265_Chuyen_Nhanh2_M" )
   END_RUNG
   // the same network as SCL:
   "AI_Pump3265_Chuyen_Nhanh2_M" := "AI_Pump3265_Chuyen_Nhanh2";
END_REGION

REGION Network 17: Mirror AI_PLC2_Me_Nhanh2_Hoan_Thanh
   RUNG wire#powerrail
      Contact( "AI_PLC2_Me_Nhanh2_Hoan_Thanh" )
      Coil( "AI_PLC2_Me_Nhanh2_Hoan_Thanh_M" )
   END_RUNG
   // the same network as SCL:
   "AI_PLC2_Me_Nhanh2_Hoan_Thanh_M" := "AI_PLC2_Me_Nhanh2_Hoan_Thanh";
END_REGION

REGION Network 18: Mirror AI_PLC2_Load_Default_Done
   RUNG wire#powerrail
      Contact( "AI_PLC2_Load_Default_Done" )
      Coil( "AI_PLC2_Load_Default_Done_M" )
   END_RUNG
   // the same network as SCL:
   "AI_PLC2_Load_Default_Done_M" := "AI_PLC2_Load_Default_Done";
END_REGION

REGION Network 19: Quyền Operator
   RUNG wire#powerrail
      Contact( "AI_HMI_Operator_Login" )
      { S7_GenerateENO := "TRUE" } Move(in := 1, out1 => "AI_HMI_User_Level")
   END_RUNG
   // the same network as SCL:
   IF "AI_HMI_Operator_Login" THEN "AI_HMI_User_Level" := 1; END_IF;
END_REGION

REGION Network 20: Quyền Engineer
   RUNG wire#powerrail
      Contact( "AI_HMI_Engineer_Login" )
      { S7_GenerateENO := "TRUE" } Move(in := 2, out1 => "AI_HMI_User_Level")
   END_RUNG
   // the same network as SCL:
   IF "AI_HMI_Engineer_Login" THEN "AI_HMI_User_Level" := 2; END_IF;
END_REGION

REGION Network 21: Quyền Admin
   RUNG wire#powerrail
      Contact( "AI_HMI_Admin_Login" )
      { S7_GenerateENO := "TRUE" } Move(in := 3, out1 => "AI_HMI_User_Level")
   END_RUNG
   // the same network as SCL:
   IF "AI_HMI_Admin_Login" THEN "AI_HMI_User_Level" := 3; END_IF;
END_REGION

REGION Network 22: Cho phép sửa thông số Engineer
   RUNG wire#powerrail
      Contact( "AI_HMI_Engineer_Login" )
      S_Coil( "AI_HMI_Cho_Phep_Sua_Thong_So" )
   END_RUNG
   // the same network as SCL:
   IF "AI_HMI_Engineer_Login" THEN "AI_HMI_Cho_Phep_Sua_Thong_So" := TRUE; END_IF;
END_REGION

REGION Network 23: Cho phép sửa thông số Admin
